LIN {X 0,Y 200.13,Z 356.551,A -85,B 0,C 180,E1 -21501.925,E2 -21501.925} C_VEL
LIN {X 0,Y 200.321,Z 356.531,A -85,B 0,C 180,E1 -21507.99,E2 -21507.99} C_VEL
LIN {X 0,Y 200.478,Z 356.509,A -85,B 0,C 180,E1 -21510,E2 -21510} C_VEL
LIN {X 0,Y 200.031,Z 356.568,A -85,B 0,C 180,E1 -21514.03,E2 -21514.03} C_VEL
LIN {X 0,Y 200.13,Z 356.553,A -85,B 0,C 180,E1 -21518.075,E2 -21518.075} C_VEL
LIN {X 0,Y 199.913,Z 356.584,A -85,B 0,C 180,E1 -21522.177,E2 -21522.177} C_VEL
LIN {X 0,Y 199.803,Z 356.594,A -85,B 0,C 180,E1 -21526.344,E2 -21526.344} C_VEL
LIN {X 0,Y 199.698,Z 356.609,A -85,B 0,C 180,E1 -21530.606,E2 -21530.606} C_VEL
LIN {X 0,Y 199.671,Z 356.608,A -85,B 0,C 180,E1 -21534.985,E2 -21534.985} C_VEL
LIN {X 0,Y 199.663,Z 356.613,A -85,B 0,C 180,E1 -21539.525,E2 -21539.525} C_VEL
LIN {X 0,Y 199.657,Z 356.613,A -85,B 0,C 180,E1 -21542.35,E2 -21542.35} C_VEL
LIN {X 0,Y 199.639,Z 356.615,A -85,B 0,C 180,E1 -21546.76,E2 -21546.76} C_VEL
LIN {X 0,Y 199.638,Z 356.616,A -85,B 0,C 180,E1 -21549.322,E2 -21549.322} C_VEL
LIN {X 0,Y 199.58,Z 356.622,A -85,B 0,C 180,E1 -21554.772,E2 -21554.772} C_VEL
LIN {X 0,Y 199.58,Z 356.626,A -85,B 0,C 180,E1 -21558.006,E2 -21558.006} C_VEL
LIN {X 0,Y 199.641,Z 356.611,A -85,B 0,C 180,E1 -21560.758,E2 -21560.758} C_VEL
LIN {X 0,Y 199.738,Z 356.771,A -85,B 0,C 180,E1 -21564.401,E2 -21564.401} C_VEL
LIN {X 0,Y 207.724,Z 383.973,A -85,B 0,C 180,E1 -21566.367,E2 -21566.367} C_VEL
LIN {X 0,Y 205.676,Z 433.557,A -85,B 0,C 180,E1 -21569.071,E2 -21569.071} C_VEL
LIN {X 0,Y 205.054,Z 449.624,A -85,B 0,C 180,E1 -21570.131,E2 -21570.131} C_VEL
LIN {X 0,Y 204.201,Z 463.538,A -85,B 0,C 180,E1 -21571.477,E2 -21571.477} C_VEL
LIN {X 0,Y 203.276,Z 475.696,A -85,B 0,C 180,E1 -21573.015,E2 -21573.015} C_VEL
LIN {X 0,Y 202.255,Z 488.035,A -85,B 0,C 180,E1 -21575.007,E2 -21575.007} C_VEL
LIN {X 0,Y 201.181,Z 499.934,A -85,B 0,C 180,E1 -21577.403,E2 -21577.403} C_VEL
LIN {X 0,Y 200.238,Z 510.281,A -85,B 0,C 180,E1 -21579.99,E2 -21579.99} C_VEL
LIN {X 0,Y 199.569,Z 519.169,A -85,B 0,C 180,E1 -21582.696,E2 -21582.696} C_VEL
LIN {X 0,Y 199.062,Z 527.201,A -85,B 0,C 180,E1 -21585.693,E2 -21585.693} C_VEL
LIN {X 0,Y 198.897,Z 534.007,A -85,B 0,C 180,E1 -21588.795,E2 -21588.795} C_VEL
LIN {X 0,Y 199.169,Z 539.493,A -85,B 0,C 180,E1 -21591.887,E2 -21591.887} C_VEL
LIN {X 0,Y 199.667,Z 543.756,A -85,B 0,C 180,E1 -21594.953,E2 -21594.953} C_VEL
LIN {X 0,Y 200.694,Z 546.982,A -85,B 0,C 180,E1 -21597.994,E2 -21597.994} C_VEL
LIN {X 0,Y 201.659,Z 548.585,A -85,B 0,C 180,E1 -21600.001,E2 -21600.001} C_VEL
LIN {X 0,Y 204.197,Z 550.567,A -85,B 0,C 180,E1 -21603.948,E2 -21603.948} C_VEL
LIN {X 0,Y 205.761,Z 550.967,A -85,B 0,C 180,E1 -21605.882,E2 -21605.882} C_VEL
LIN {X 0,Y 207.575,Z 550.921,A -85,B 0,C 180,E1 -21607.784,E2 -21607.784} C_VEL
LIN {X 0,Y 211.909,Z 549.645,A -85,B 0,C 180,E1 -21611.479,E2 -21611.479} C_VEL
LIN {X 0,Y 214.316,Z 548.421,A -85,B 0,C 180,E1 -21613.271,E2 -21613.271} C_VEL
LIN {X 0,Y 218.335,Z 545.769,A -85,B 0,C 180,E1 -21615.88,E2 -21615.88} C_VEL
LIN {X 0,Y 224.368,Z 540.635,A -85,B 0,C 180,E1 -21619.203,E2 -21619.203} C_VEL
LIN {X 0,Y 230.212,Z 534.494,A -85,B 0,C 180,E1 -21621.962,E2 -21621.962} C_VEL
LIN {X 0,Y 235.618,Z 527.868,A -85,B 0,C 180,E1 -21624.214,E2 -21624.214} C_VEL
LIN {X 0,Y 241.34,Z 519.724,A -85,B 0,C 180,E1 -21626.366,E2 -21626.366} C_VEL
LIN {X 0,Y 247.352,Z 509.665,A -85,B 0,C 180,E1 -21628.42,E2 -21628.42} C_VEL
LIN {X 0,Y 252.531,Z 499.378,A -85,B 0,C 180,E1 -21630.063,E2 -21630.063} C_VEL
LIN {X 0,Y 257.926,Z 486.52,A -85,B 0,C 180,E1 -21631.637,E2 -21631.637} C_VEL
LIN {X 0,Y 262.112,Z 473.808,A -85,B 0,C 180,E1 -21632.857,E2 -21632.857} C_VEL
LIN {X 0,Y 265.465,Z 460.103,A -85,B 0,C 180,E1 -21633.86,E2 -21633.86} C_VEL
LIN {X 0,Y 269.789,Z 438.336,A -85,B 0,C 180,E1 -21635.008,E2 -21635.008} C_VEL
LIN {X 0,Y 269.332,Z 436.976,A -85,B 0,C 180,E1 -21636.008,E2 -21636.008} C_VEL
LIN {X 0,Y 268.866,Z 435.366,A -85,B 0,C 180,E1 -21637.692,E2 -21637.692} C_VEL
LIN {X 0,Y 268.411,Z 435.595,A -85,B 0,C 180,E1 -21639.946,E2 -21639.946} C_VEL
LIN {X 0,Y 268.781,Z 437.514,A -85,B 0,C 180,E1 -21642.832,E2 -21642.832} C_VEL
LIN {X 0,Y 268.989,Z 439.1,A -85,B 0,C 180,E1 -21643.838,E2 -21643.838} C_VEL
LIN {X 0,Y 266.129,Z 456.669,A -85,B 0,C 180,E1 -21645.491,E2 -21645.491} C_VEL
LIN {X 0,Y 265.42,Z 460.479,A -85,B 0,C 180,E1 -21645.712,E2 -21645.712} C_VEL
LIN {X 0,Y 264.093,Z 466.352,A -85,B 0,C 180,E1 -21645.82,E2 -21645.82} C_VEL
LIN {X 0,Y 259.559,Z 481.708,A -85,B 0,C 180,E1 -21645.699,E2 -21645.699} C_VEL
LIN {X 0,Y 257.716,Z 487.218,A -85,B 0,C 180,E1 -21645.861,E2 -21645.861} C_VEL
LIN {X 0,Y 252.173,Z 502.361,A -85,B 0,C 180,E1 -21646.81,E2 -21646.81} C_VEL
LIN {X 0,Y 246.736,Z 514.517,A -85,B 0,C 180,E1 -21647.816,E2 -21647.816} C_VEL
LIN {X 0,Y 240.342,Z 526.637,A -85,B 0,C 180,E1 -21649.134,E2 -21649.134} C_VEL
LIN {X 0,Y 233.392,Z 538.193,A -85,B 0,C 180,E1 -21650.775,E2 -21650.775} C_VEL
LIN {X 0,Y 226.298,Z 548.528,A -85,B 0,C 180,E1 -21652.727,E2 -21652.727} C_VEL
LIN {X 0,Y 219.772,Z 557.196,A -85,B 0,C 180,E1 -21654.857,E2 -21654.857} C_VEL
LIN {X 0,Y 212.934,Z 565.506,A -85,B 0,C 180,E1 -21657.565,E2 -21657.565} C_VEL
LIN {X 0,Y 207.028,Z 572.262,A -85,B 0,C 180,E1 -21660.512,E2 -21660.512} C_VEL
LIN {X 0,Y 201.244,Z 578.3,A -85,B 0,C 180,E1 -21664.116,E2 -21664.116} C_VEL
LIN {X 0,Y 197.743,Z 581.793,A -85,B 0,C 180,E1 -21666.986,E2 -21666.986} C_VEL
LIN {X 0,Y 194.328,Z 585.191,A -85,B 0,C 180,E1 -21671.004,E2 -21671.004} C_VEL
LIN {X 0,Y 192.114,Z 587.173,A -85,B 0,C 180,E1 -21675.162,E2 -21675.162} C_VEL
LIN {X 0,Y 191.331,Z 587.716,A -85,B 0,C 180,E1 -21679.417,E2 -21679.417} C_VEL
LIN {X 0,Y 191.839,Z 586.864,A -85,B 0,C 180,E1 -21683.69,E2 -21683.69} C_VEL
LIN {X 0,Y 192.41,Z 585.854,A -85,B 0,C 180,E1 -21685.81,E2 -21685.81} C_VEL
LIN {X 0,Y 193.156,Z 584.419,A -85,B 0,C 180,E1 -21687.914,E2 -21687.914} C_VEL
LIN {X 0,Y 194.107,Z 581.798,A -85,B 0,C 180,E1 -21690.778,E2 -21690.778} C_VEL
LIN {X 0,Y 192.821,Z 584.818,A -85,B 0,C 180,E1 -21694.18,E2 -21694.18} C_VEL
LIN {X 0,Y 191.765,Z 586.935,A -85,B 0,C 180,E1 -21698.429,E2 -21698.429} C_VEL
LIN {X 0,Y 191.724,Z 587.605,A -85,B 0,C 180,E1 -21702.705,E2 -21702.705} C_VEL
LIN {X 0,Y 193.151,Z 586.968,A -85,B 0,C 180,E1 -21706.923,E2 -21706.923} C_VEL
LIN {X 0,Y 196.036,Z 584.878,A -85,B 0,C 180,E1 -21711.231,E2 -21711.231} C_VEL
LIN {X 0,Y 200.066,Z 581.723,A -85,B 0,C 180,E1 -21714.932,E2 -21714.932} C_VEL
LIN {X 0,Y 205.555,Z 577.043,A -85,B 0,C 180,E1 -21718.598,E2 -21718.598} C_VEL
LIN {X 0,Y 212.272,Z 570.882,A -85,B 0,C 180,E1 -21721.987,E2 -21721.987} C_VEL
LIN {X 0,Y 219.024,Z 564.138,A -85,B 0,C 180,E1 -21724.719,E2 -21724.719} C_VEL
LIN {X 0,Y 226.551,Z 555.909,A -85,B 0,C 180,E1 -21727.223,E2 -21727.223} C_VEL
LIN {X 0,Y 233.695,Z 547.449,A -85,B 0,C 180,E1 -21729.164,E2 -21729.164} C_VEL
LIN {X 0,Y 241.357,Z 537.432,A -85,B 0,C 180,E1 -21730.934,E2 -21730.934} C_VEL
LIN {X 0,Y 249.417,Z 525.489,A -85,B 0,C 180,E1 -21732.552,E2 -21732.552} C_VEL
LIN {X 0,Y 256.63,Z 513.371,A -85,B 0,C 180,E1 -21733.748,E2 -21733.748} C_VEL
LIN {X 0,Y 263.345,Z 500.187,A -85,B 0,C 180,E1 -21734.739,E2 -21734.739} C_VEL
LIN {X 0,Y 269.568,Z 485.453,A -85,B 0,C 180,E1 -21735.585,E2 -21735.585} C_VEL
LIN {X 0,Y 274.038,Z 472.123,A -85,B 0,C 180,E1 -21736.246,E2 -21736.246} C_VEL
LIN {X 0,Y 276.158,Z 464.301,A -85,B 0,C 180,E1 -21736.993,E2 -21736.993} C_VEL
LIN {X 0,Y 276.362,Z 463.489,A -85,B 0,C 180,E1 -21737.517,E2 -21737.517} C_VEL
LIN {X 0,Y 276.331,Z 463.603,A -85,B 0,C 180,E1 -21737.696,E2 -21737.696} C_VEL
LIN {X 0,Y 272.737,Z 475.349,A -85,B 0,C 180,E1 -21738.477,E2 -21738.477} C_VEL
LIN {X 0,Y 268.039,Z 487.452,A -85,B 0,C 180,E1 -21739.498,E2 -21739.498} C_VEL
LIN {X 0,Y 262.451,Z 499.125,A -85,B 0,C 180,E1 -21740.754,E2 -21740.754} C_VEL
LIN {X 0,Y 257,Z 508.731,A -85,B 0,C 180,E1 -21742.026,E2 -21742.026} C_VEL
LIN {X 0,Y 249.982,Z 519.179,A -85,B 0,C 180,E1 -21743.814,E2 -21743.814} C_VEL
LIN {X 0,Y 243.171,Z 527.827,A -85,B 0,C 180,E1 -21745.695,E2 -21745.695} C_VEL
LIN {X 0,Y 235.644,Z 535.955,A -85,B 0,C 180,E1 -21748.035,E2 -21748.035} C_VEL
LIN {X 0,Y 228.609,Z 542.34,A -85,B 0,C 180,E1 -21750.535,E2 -21750.535} C_VEL
LIN {X 0,Y 222.953,Z 546.638,A -85,B 0,C 180,E1 -21752.801,E2 -21752.801} C_VEL
LIN {X 0,Y 217.696,Z 549.945,A -85,B 0,C 180,E1 -21755.184,E2 -21755.184} C_VEL
LIN {X 0,Y 211.361,Z 552.899,A -85,B 0,C 180,E1 -21758.545,E2 -21758.545} C_VEL
LIN {X 0,Y 208.492,Z 553.807,A -85,B 0,C 180,E1 -21760.3,E2 -21760.3} C_VEL
LIN {X 0,Y 203.337,Z 554.428,A -85,B 0,C 180,E1 -21763.947,E2 -21763.947} C_VEL
LIN {X 0,Y 199.159,Z 553.524,A -85,B 0,C 180,E1 -21767.775,E2 -21767.775} C_VEL
LIN {X 0,Y 197.465,Z 552.5,A -85,B 0,C 180,E1 -21769.748,E2 -21769.748} C_VEL
LIN {X 0,Y 194.698,Z 549.233,A -85,B 0,C 180,E1 -21773.782,E2 -21773.782} C_VEL
LIN {X 0,Y 192.883,Z 544.368,A -85,B 0,C 180,E1 -21777.911,E2 -21777.911} C_VEL
LIN {X 0,Y 192.027,Z 539.501,A -85,B 0,C 180,E1 -21781.048,E2 -21781.048} C_VEL
LIN {X 0,Y 191.753,Z 532.354,A -85,B 0,C 180,E1 -21784.729,E2 -21784.729} C_VEL
LIN {X 0,Y 191.932,Z 526.232,A -85,B 0,C 180,E1 -21787.335,E2 -21787.335} C_VEL
LIN {X 0,Y 192.376,Z 517.232,A -85,B 0,C 180,E1 -21790.524,E2 -21790.524} C_VEL
LIN {X 0,Y 193.015,Z 507.213,A -85,B 0,C 180,E1 -21793.421,E2 -21793.421} C_VEL
LIN {X 0,Y 193.977,Z 494.938,A -85,B 0,C 180,E1 -21796.306,E2 -21796.306} C_VEL
LIN {X 0,Y 194.877,Z 482.252,A -85,B 0,C 180,E1 -21798.666,E2 -21798.666} C_VEL
LIN {X 0,Y 195.949,Z 469.152,A -85,B 0,C 180,E1 -21800.605,E2 -21800.605} C_VEL
LIN {X 0,Y 196.739,Z 454.506,A -85,B 0,C 180,E1 -21802.263,E2 -21802.263} C_VEL
LIN {X 0,Y 197.458,Z 440.483,A -85,B 0,C 180,E1 -21803.395,E2 -21803.395} C_VEL
LIN {X 0,Y 199.499,Z 382.365,A -85,B 0,C 180,E1 -21806.992,E2 -21806.992} C_VEL
LIN {X 0,Y 192.727,Z 357.475,A -85,B 0,C 180,E1 -21808.874,E2 -21808.874} C_VEL
LIN {X 0,Y 192.598,Z 357.494,A -85,B 0,C 180,E1 -21813.185,E2 -21813.185} C_VEL
LIN {X 0,Y 192.55,Z 357.496,A -85,B 0,C 180,E1 -21818.351,E2 -21818.351} C_VEL
LIN {X 0,Y 192.49,Z 357.507,A -85,B 0,C 180,E1 -21823.095,E2 -21823.095} C_VEL
LIN {X 0,Y 192.513,Z 357.501,A -85,B 0,C 180,E1 -21826.896,E2 -21826.896} C_VEL
LIN {X 0,Y 192.572,Z 357.496,A -85,B 0,C 180,E1 -21831.653,E2 -21831.653} C_VEL
LIN {X 0,Y 192.596,Z 357.493,A -85,B 0,C 180,E1 -21834.278,E2 -21834.278} C_VEL
LIN {X 0,Y 192.597,Z 357.493,A -85,B 0,C 180,E1 -21839.278,E2 -21839.278} C_VEL
LIN {X 0,Y 192.658,Z 357.484,A -85,B 0,C 180,E1 -21841.691,E2 -21841.691} C_VEL
LIN {X 0,Y 192.703,Z 357.479,A -85,B 0,C 180,E1 -21846.349,E2 -21846.349} C_VEL
LIN {X 0,Y 192.729,Z 357.474,A -85,B 0,C 180,E1 -21851.457,E2 -21851.457} C_VEL
LIN {X 0,Y 192.77,Z 357.471,A -85,B 0,C 180,E1 -21855.214,E2 -21855.214} C_VEL
LIN {X 0,Y 193.018,Z 357.439,A -85,B 0,C 180,E1 -21859.511,E2 -21859.511} C_VEL
LIN {X 0,Y 193.003,Z 357.441,A -85,B 0,C 180,E1 -21863.729,E2 -21863.729} C_VEL
LIN {X 0,Y 193.263,Z 357.41,A -85,B 0,C 180,E1 -21867.916,E2 -21867.916} C_VEL
LIN {X 0,Y 193.442,Z 357.385,A -85,B 0,C 180,E1 -21870,E2 -21870} C_VEL
LIN {X 0,Y 192.978,Z 357.447,A -85,B 0,C 180,E1 -21874.177,E2 -21874.177} C_VEL
LIN {X 0,Y 193.077,Z 357.431,A -85,B 0,C 180,E1 -21878.372,E2 -21878.372} C_VEL
LIN {X 0,Y 192.852,Z 357.462,A -85,B 0,C 180,E1 -21882.63,E2 -21882.63} C_VEL
LIN {X 0,Y 192.756,Z 357.469,A -85,B 0,C 180,E1 -21886.959,E2 -21886.959} C_VEL
LIN {X 0,Y 192.635,Z 357.488,A -85,B 0,C 180,E1 -21891.398,E2 -21891.398} C_VEL
LIN {X 0,Y 192.663,Z 357.484,A -85,B 0,C 180,E1 -21894.225,E2 -21894.225} C_VEL
LIN {X 0,Y 192.643,Z 357.487,A -85,B 0,C 180,E1 -21898.89,E2 -21898.89} C_VEL
LIN {X 0,Y 192.597,Z 357.49,A -85,B 0,C 180,E1 -21903.187,E2 -21903.187} C_VEL
LIN {X 0,Y 192.609,Z 357.492,A -85,B 0,C 180,E1 -21906.609,E2 -21906.609} C_VEL
LIN {X 0,Y 192.523,Z 357.5,A -85,B 0,C 180,E1 -21911.079,E2 -21911.079} C_VEL
LIN {X 0,Y 192.512,Z 357.506,A -85,B 0,C 180,E1 -21916.083,E2 -21916.083} C_VEL
LIN {X 0,Y 192.54,Z 357.499,A -85,B 0,C 180,E1 -21920.044,E2 -21920.044} C_VEL
LIN {X 0,Y 192.649,Z 357.488,A -85,B 0,C 180,E1 -21923.981,E2 -21923.981} C_VEL
LIN {X 0,Y 200.688,Z 384.623,A -85,B 0,C 180,E1 -21926.079,E2 -21926.079} C_VEL
LIN {X 0,Y 198.622,Z 434.427,A -85,B 0,C 180,E1 -21928.911,E2 -21928.911} C_VEL
LIN {X 0,Y 197.991,Z 450.137,A -85,B 0,C 180,E1 -21929.983,E2 -21929.983} C_VEL
LIN {X 0,Y 197.112,Z 464.132,A -85,B 0,C 180,E1 -21931.374,E2 -21931.374} C_VEL
LIN {X 0,Y 196.156,Z 476.48,A -85,B 0,C 180,E1 -21932.99,E2 -21932.99} C_VEL
LIN {X 0,Y 195.142,Z 488.274,A -85,B 0,C 180,E1 -21934.966,E2 -21934.966} C_VEL
LIN {X 0,Y 194.09,Z 499.915,A -85,B 0,C 180,E1 -21937.374,E2 -21937.374} C_VEL
LIN {X 0,Y 193.057,Z 511.324,A -85,B 0,C 180,E1 -21940.323,E2 -21940.323} C_VEL
LIN {X 0,Y 192.414,Z 519.875,A -85,B 0,C 180,E1 -21943.011,E2 -21943.011} C_VEL
LIN {X 0,Y 191.935,Z 528.245,A -85,B 0,C 180,E1 -21946.232,E2 -21946.232} C_VEL
LIN {X 0,Y 191.846,Z 535.03,A -85,B 0,C 180,E1 -21949.447,E2 -21949.447} C_VEL
LIN {X 0,Y 192.176,Z 540.475,A -85,B 0,C 180,E1 -21952.647,E2 -21952.647} C_VEL
LIN {X 0,Y 192.784,Z 544.764,A -85,B 0,C 180,E1 -21955.82,E2 -21955.82} C_VEL
LIN {X 0,Y 193.516,Z 547.04,A -85,B 0,C 180,E1 -21957.92,E2 -21957.92} C_VEL
LIN {X 0,Y 194.508,Z 548.879,A -85,B 0,C 180,E1 -21960.001,E2 -21960.001} C_VEL
LIN {X 0,Y 195.68,Z 550.312,A -85,B 0,C 180,E1 -21962.059,E2 -21962.059} C_VEL
LIN {X 0,Y 197.384,Z 551.462,A -85,B 0,C 180,E1 -21964.459,E2 -21964.459} C_VEL
LIN {X 0,Y 200.579,Z 552.142,A -85,B 0,C 180,E1 -21968.058,E2 -21968.058} C_VEL
LIN {X 0,Y 202.729,Z 551.962,A -85,B 0,C 180,E1 -21969.983,E2 -21969.983} C_VEL
LIN {X 0,Y 205.076,Z 551.368,A -85,B 0,C 180,E1 -21971.867,E2 -21971.867} C_VEL
LIN {X 0,Y 210.303,Z 548.958,A -85,B 0,C 180,E1 -21975.507,E2 -21975.507} C_VEL
LIN {X 0,Y 213.822,Z 546.747,A -85,B 0,C 180,E1 -21977.599,E2 -21977.599} C_VEL
LIN {X 0,Y 219.704,Z 542.124,A -85,B 0,C 180,E1 -21980.603,E2 -21980.603} C_VEL
LIN {X 0,Y 225.014,Z 537.117,A -85,B 0,C 180,E1 -21982.982,E2 -21982.982} C_VEL
LIN {X 0,Y 230.666,Z 530.851,A -85,B 0,C 180,E1 -21985.25,E2 -21985.25} C_VEL
LIN {X 0,Y 237.701,Z 521.712,A -85,B 0,C 180,E1 -21987.755,E2 -21987.755} C_VEL
LIN {X 0,Y 242.961,Z 513.651,A -85,B 0,C 180,E1 -21989.456,E2 -21989.456} C_VEL
LIN {X 0,Y 249.252,Z 502.412,A -85,B 0,C 180,E1 -21991.329,E2 -21991.329} C_VEL
LIN {X 0,Y 254.572,Z 490.786,A -85,B 0,C 180,E1 -21992.806,E2 -21992.806} C_VEL
LIN {X 0,Y 259.07,Z 478.805,A -85,B 0,C 180,E1 -21994.023,E2 -21994.023} C_VEL
LIN {X 0,Y 262.899,Z 465.581,A -85,B 0,C 180,E1 -21995.049,E2 -21995.049} C_VEL
LIN {X 0,Y 266.056,Z 450.737,A -85,B 0,C 180,E1 -21995.915,E2 -21995.915} C_VEL
LIN {X 0,Y 267.539,Z 443.724,A -85,B 0,C 180,E1 -21996.288,E2 -21996.288} C_VEL
LIN {X 0,Y 267.125,Z 442.24,A -85,B 0,C 180,E1 -21997.88,E2 -21997.88} C_VEL
LIN {X 0,Y 266.747,Z 442.503,A -85,B 0,C 180,E1 -21999.886,E2 -21999.886} C_VEL
LIN {X 0,Y 266.995,Z 444.365,A -85,B 0,C 180,E1 -22002.597,E2 -22002.597} C_VEL
LIN {X 0,Y 267.021,Z 444.576,A -85,B 0,C 180,E1 -22002.741,E2 -22002.741} C_VEL
LIN {X 0,Y 263.718,Z 462.474,A -85,B 0,C 180,E1 -22004.399,E2 -22004.399} C_VEL
LIN {X 0,Y 261.617,Z 473.4,A -85,B 0,C 180,E1 -22005.177,E2 -22005.177} C_VEL
LIN {X 0,Y 257.716,Z 487.218,A -85,B 0,C 180,E1 -22005.861,E2 -22005.861} C_VEL
LIN {X 0,Y 255.648,Z 492.809,A -85,B 0,C 180,E1 -22006.03,E2 -22006.03} C_VEL
LIN {X 0,Y 251.391,Z 501.746,A -85,B 0,C 180,E1 -22005.971,E2 -22005.971} C_VEL
LIN {X 0,Y 246.689,Z 510.398,A -85,B 0,C 180,E1 -22005.995,E2 -22005.995} C_VEL
LIN {X 0,Y 243.93,Z 515.393,A -85,B 0,C 180,E1 -22006.303,E2 -22006.303} C_VEL
LIN {X 0,Y 236.508,Z 528.466,A -85,B 0,C 180,E1 -22007.753,E2 -22007.753} C_VEL
LIN {X 0,Y 229.335,Z 539.311,A -85,B 0,C 180,E1 -22009.367,E2 -22009.367} C_VEL
LIN {X 0,Y 221.989,Z 549.224,A -85,B 0,C 180,E1 -22011.297,E2 -22011.297} C_VEL
LIN {X 0,Y 215.177,Z 557.482,A -85,B 0,C 180,E1 -22013.41,E2 -22013.41} C_VEL
LIN {X 0,Y 207.967,Z 565.461,A -85,B 0,C 180,E1 -22016.11,E2 -22016.11} C_VEL
LIN {X 0,Y 200.902,Z 572.726,A -85,B 0,C 180,E1 -22019.519,E2 -22019.519} C_VEL
LIN {X 0,Y 196.268,Z 577.061,A -85,B 0,C 180,E1 -22022.256,E2 -22022.256} C_VEL
LIN {X 0,Y 191.203,Z 581.517,A -85,B 0,C 180,E1 -22026.151,E2 -22026.151} C_VEL
LIN {X 0,Y 187.601,Z 584.519,A -85,B 0,C 180,E1 -22030.295,E2 -22030.295} C_VEL
LIN {X 0,Y 185.248,Z 586.153,A -85,B 0,C 180,E1 -22034.599,E2 -22034.599} C_VEL
LIN {X 0,Y 184.37,Z 586.445,A -85,B 0,C 180,E1 -22039.012,E2 -22039.012} C_VEL
LIN {X 0,Y 184.867,Z 585.307,A -85,B 0,C 180,E1 -22043.451,E2 -22043.451} C_VEL
LIN {X 0,Y 185.473,Z 584.166,A -85,B 0,C 180,E1 -22045.653,E2 -22045.653} C_VEL
LIN {X 0,Y 186.656,Z 581.612,A -85,B 0,C 180,E1 -22048.921,E2 -22048.921} C_VEL
LIN {X 0,Y 187.358,Z 579.59,A -85,B 0,C 180,E1 -22050.806,E2 -22050.806} C_VEL
LIN {X 0,Y 185.971,Z 582.827,A -85,B 0,C 180,E1 -22054.334,E2 -22054.334} C_VEL
LIN {X 0,Y 184.847,Z 585.245,A -85,B 0,C 180,E1 -22058.747,E2 -22058.747} C_VEL
LIN {X 0,Y 184.846,Z 586.225,A -85,B 0,C 180,E1 -22063.186,E2 -22063.186} C_VEL
LIN {X 0,Y 186.365,Z 585.91,A -85,B 0,C 180,E1 -22067.559,E2 -22067.559} C_VEL
LIN {X 0,Y 189.237,Z 584.289,A -85,B 0,C 180,E1 -22071.801,E2 -22071.801} C_VEL
LIN {X 0,Y 193.651,Z 581.401,A -85,B 0,C 180,E1 -22075.817,E2 -22075.817} C_VEL
LIN {X 0,Y 199.364,Z 577.196,A -85,B 0,C 180,E1 -22079.573,E2 -22079.573} C_VEL
LIN {X 0,Y 206.32,Z 571.582,A -85,B 0,C 180,E1 -22083.026,E2 -22083.026} C_VEL
LIN {X 0,Y 214.334,Z 564.352,A -85,B 0,C 180,E1 -22086.172,E2 -22086.172} C_VEL
LIN {X 0,Y 222.215,Z 556.563,A -85,B 0,C 180,E1 -22088.655,E2 -22088.655} C_VEL
LIN {X 0,Y 229.62,Z 548.574,A -85,B 0,C 180,E1 -22090.572,E2 -22090.572} C_VEL
LIN {X 0,Y 237.681,Z 538.972,A -85,B 0,C 180,E1 -22092.333,E2 -22092.333} C_VEL
LIN {X 0,Y 246.54,Z 526.919,A -85,B 0,C 180,E1 -22094.015,E2 -22094.015} C_VEL
LIN {X 0,Y 253.958,Z 515.491,A -85,B 0,C 180,E1 -22095.165,E2 -22095.165} C_VEL
LIN {X 0,Y 261.65,Z 501.585,A -85,B 0,C 180,E1 -22096.209,E2 -22096.209} C_VEL
LIN {X 0,Y 268.087,Z 487.622,A -85,B 0,C 180,E1 -22097.002,E2 -22097.002} C_VEL
LIN {X 0,Y 269.692,Z 483.656,A -85,B 0,C 180,E1 -22097.198,E2 -22097.198} C_VEL
LIN {X 0,Y 270.146,Z 482.401,A -85,B 0,C 180,E1 -22097.436,E2 -22097.436} C_VEL
LIN {X 0,Y 264.358,Z 495.071,A -85,B 0,C 180,E1 -22098.6,E2 -22098.6} C_VEL
LIN {X 0,Y 257.994,Z 506.481,A -85,B 0,C 180,E1 -22099.941,E2 -22099.941} C_VEL
LIN {X 0,Y 251.328,Z 516.468,A -85,B 0,C 180,E1 -22101.459,E2 -22101.459} C_VEL
LIN {X 0,Y 243.909,Z 525.948,A -85,B 0,C 180,E1 -22103.28,E2 -22103.28} C_VEL
LIN {X 0,Y 236.936,Z 533.527,A -85,B 0,C 180,E1 -22105.179,E2 -22105.179} C_VEL
LIN {X 0,Y 229.184,Z 540.728,A -85,B 0,C 180,E1 -22107.544,E2 -22107.544} C_VEL
LIN {X 0,Y 220.945,Z 546.965,A -85,B 0,C 180,E1 -22110.459,E2 -22110.459} C_VEL
LIN {X 0,Y 215.201,Z 550.488,A -85,B 0,C 180,E1 -22112.792,E2 -22112.792} C_VEL
LIN {X 0,Y 211.587,Z 552.337,A -85,B 0,C 180,E1 -22114.417,E2 -22114.417} C_VEL
LIN {X 0,Y 208.165,Z 553.761,A -85,B 0,C 180,E1 -22116.099,E2 -22116.099} C_VEL
LIN {X 0,Y 201.997,Z 555.423,A -85,B 0,C 180,E1 -22119.639,E2 -22119.639} C_VEL
LIN {X 0,Y 196.63,Z 555.631,A -85,B 0,C 180,E1 -22123.384,E2 -22123.384} C_VEL
LIN {X 0,Y 192.261,Z 554.259,A -85,B 0,C 180,E1 -22127.329,E2 -22127.329} C_VEL
LIN {X 0,Y 188.969,Z 551.386,A -85,B 0,C 180,E1 -22131.444,E2 -22131.444} C_VEL
LIN {X 0,Y 187.103,Z 548.173,A -85,B 0,C 180,E1 -22134.611,E2 -22134.611} C_VEL
LIN {X 0,Y 185.795,Z 544.013,A -85,B 0,C 180,E1 -22137.831,E2 -22137.831} C_VEL
LIN {X 0,Y 184.928,Z 538.801,A -85,B 0,C 180,E1 -22141.088,E2 -22141.088} C_VEL
LIN {X 0,Y 184.707,Z 531.242,A -85,B 0,C 180,E1 -22144.91,E2 -22144.91} C_VEL
LIN {X 0,Y 184.913,Z 523.993,A -85,B 0,C 180,E1 -22147.908,E2 -22147.908} C_VEL
LIN {X 0,Y 185.411,Z 515.207,A -85,B 0,C 180,E1 -22150.924,E2 -22150.924} C_VEL
LIN {X 0,Y 186.063,Z 504.602,A -85,B 0,C 180,E1 -22153.933,E2 -22153.933} C_VEL
LIN {X 0,Y 187.02,Z 492.722,A -85,B 0,C 180,E1 -22156.65,E2 -22156.65} C_VEL
LIN {X 0,Y 187.882,Z 481.063,A -85,B 0,C 180,E1 -22158.821,E2 -22158.821} C_VEL
LIN {X 0,Y 188.946,Z 467.407,A -85,B 0,C 180,E1 -22160.834,E2 -22160.834} C_VEL
LIN {X 0,Y 189.688,Z 453.534,A -85,B 0,C 180,E1 -22162.389,E2 -22162.389} C_VEL
LIN {X 0,Y 190.415,Z 439.593,A -85,B 0,C 180,E1 -22163.519,E2 -22163.519} C_VEL
LIN {X 0,Y 192.431,Z 383.401,A -85,B 0,C 180,E1 -22167.166,E2 -22167.166} C_VEL
LIN {X 0,Y 185.653,Z 358.355,A -85,B 0,C 180,E1 -22169.104,E2 -22169.104} C_VEL
LIN {X 0,Y 185.498,Z 358.379,A -85,B 0,C 180,E1 -22174.631,E2 -22174.631} C_VEL
LIN {X 0,Y 185.504,Z 358.374,A -85,B 0,C 180,E1 -22177.312,E2 -22177.312} C_VEL
LIN {X 0,Y 185.47,Z 358.381,A -85,B 0,C 180,E1 -22180.724,E2 -22180.724} C_VEL
LIN {X 0,Y 185.48,Z 358.377,A -85,B 0,C 180,E1 -22186.047,E2 -22186.047} C_VEL
LIN {X 0,Y 185.487,Z 358.378,A -85,B 0,C 180,E1 -22189.901,E2 -22189.901} C_VEL
LIN {X 0,Y 185.541,Z 358.373,A -85,B 0,C 180,E1 -22192.695,E2 -22192.695} C_VEL
LIN {X 0,Y 185.538,Z 358.371,A -85,B 0,C 180,E1 -22197.974,E2 -22197.974} C_VEL
LIN {X 0,Y 185.578,Z 358.37,A -85,B 0,C 180,E1 -22200.576,E2 -22200.576} C_VEL
LIN {X 0,Y 185.585,Z 358.364,A -85,B 0,C 180,E1 -22205.382,E2 -22205.382} C_VEL
LIN {X 0,Y 185.605,Z 358.364,A -85,B 0,C 180,E1 -22210.075,E2 -22210.075} C_VEL
LIN {X 0,Y 185.722,Z 358.35,A -85,B 0,C 180,E1 -22214.64,E2 -22214.64} C_VEL
LIN {X 0,Y 185.94,Z 358.32,A -85,B 0,C 180,E1 -22219.328,E2 -22219.328} C_VEL
LIN {X 0,Y 185.967,Z 358.317,A -85,B 0,C 180,E1 -22223.49,E2 -22223.49} C_VEL
LIN {X 0,Y 186.207,Z 358.288,A -85,B 0,C 180,E1 -22227.837,E2 -22227.837} C_VEL
LIN {X 0,Y 186.405,Z 358.261,A -85,B 0,C 180,E1 -22230,E2 -22230} C_VEL
LIN {X 0,Y 185.926,Z 358.327,A -85,B 0,C 180,E1 -22234.336,E2 -22234.336} C_VEL
LIN {X 0,Y 186.027,Z 358.309,A -85,B 0,C 180,E1 -22238.692,E2 -22238.692} C_VEL
LIN {X 0,Y 185.763,Z 358.344,A -85,B 0,C 180,E1 -22243.121,E2 -22243.121} C_VEL
LIN {X 0,Y 185.688,Z 358.349,A -85,B 0,C 180,E1 -22247.626,E2 -22247.626} C_VEL
LIN {X 0,Y 185.595,Z 358.367,A -85,B 0,C 180,E1 -22252.252,E2 -22252.252} C_VEL
LIN {X 0,Y 185.559,Z 358.368,A -85,B 0,C 180,E1 -22257.033,E2 -22257.033} C_VEL
LIN {X 0,Y 185.576,Z 358.368,A -85,B 0,C 180,E1 -22259.494,E2 -22259.494} C_VEL
LIN {X 0,Y 185.517,Z 358.373,A -85,B 0,C 180,E1 -22264.629,E2 -22264.629} C_VEL
LIN {X 0,Y 185.543,Z 358.371,A -85,B 0,C 180,E1 -22267.305,E2 -22267.305} C_VEL
LIN {X 0,Y 185.485,Z 358.377,A -85,B 0,C 180,E1 -22270.731,E2 -22270.731} C_VEL
LIN {X 0,Y 185.478,Z 358.382,A -85,B 0,C 180,E1 -22276.05,E2 -22276.05} C_VEL
LIN {X 0,Y 185.488,Z 358.378,A -85,B 0,C 180,E1 -22279.902,E2 -22279.902} C_VEL
LIN {X 0,Y 185.63,Z 358.433,A -85,B 0,C 180,E1 -22283.681,E2 -22283.681} C_VEL
LIN {X 0,Y 193.594,Z 386.068,A -85,B 0,C 180,E1 -22285.823,E2 -22285.823} C_VEL
LIN {X 0,Y 191.303,Z 441.155,A -85,B 0,C 180,E1 -22289.126,E2 -22289.126} C_VEL
LIN {X 0,Y 190.593,Z 455.398,A -85,B 0,C 180,E1 -22290.298,E2 -22290.298} C_VEL
LIN {X 0,Y 189.683,Z 469.139,A -85,B 0,C 180,E1 -22291.871,E2 -22291.871} C_VEL
LIN {X 0,Y 188.63,Z 481.707,A -85,B 0,C 180,E1 -22293.741,E2 -22293.741} C_VEL
LIN {X 0,Y 187.552,Z 493.474,A -85,B 0,C 180,E1 -22295.953,E2 -22295.953} C_VEL
LIN {X 0,Y 186.55,Z 504.298,A -85,B 0,C 180,E1 -22298.451,E2 -22298.451} C_VEL
LIN {X 0,Y 185.707,Z 514.647,A -85,B 0,C 180,E1 -22301.38,E2 -22301.38} C_VEL
LIN {X 0,Y 185.082,Z 523.842,A -85,B 0,C 180,E1 -22304.586,E2 -22304.586} C_VEL
LIN {X 0,Y 184.749,Z 531.604,A -85,B 0,C 180,E1 -22307.924,E2 -22307.924} C_VEL
LIN {X 0,Y 184.919,Z 537.913,A -85,B 0,C 180,E1 -22311.257,E2 -22311.257} C_VEL
LIN {X 0,Y 185.368,Z 542.985,A -85,B 0,C 180,E1 -22314.562,E2 -22314.562} C_VEL
LIN {X 0,Y 186.341,Z 546.938,A -85,B 0,C 180,E1 -22317.84,E2 -22317.84} C_VEL
LIN {X 0,Y 187.348,Z 549.033,A -85,B 0,C 180,E1 -22320.001,E2 -22320.001} C_VEL
LIN {X 0,Y 188.546,Z 550.705,A -85,B 0,C 180,E1 -22322.137,E2 -22322.137} C_VEL
LIN {X 0,Y 191.679,Z 552.789,A -85,B 0,C 180,E1 -22326.316,E2 -22326.316} C_VEL
LIN {X 0,Y 193.578,Z 553.264,A -85,B 0,C 180,E1 -22328.351,E2 -22328.351} C_VEL
LIN {X 0,Y 195.799,Z 553.306,A -85,B 0,C 180,E1 -22330.34,E2 -22330.34} C_VEL
LIN {X 0,Y 200.853,Z 552.197,A -85,B 0,C 180,E1 -22334.179,E2 -22334.179} C_VEL
LIN {X 0,Y 203.676,Z 551.088,A -85,B 0,C 180,E1 -22336.025,E2 -22336.025} C_VEL
LIN {X 0,Y 206.703,Z 549.524,A -85,B 0,C 180,E1 -22337.82,E2 -22337.82} C_VEL
LIN {X 0,Y 213.406,Z 545.132,A -85,B 0,C 180,E1 -22341.24,E2 -22341.24} C_VEL
LIN {X 0,Y 218.914,Z 540.596,A -85,B 0,C 180,E1 -22343.66,E2 -22343.66} C_VEL
LIN {X 0,Y 225.783,Z 533.837,A -85,B 0,C 180,E1 -22346.332,E2 -22346.332} C_VEL
LIN {X 0,Y 232.005,Z 526.651,A -85,B 0,C 180,E1 -22348.449,E2 -22348.449} C_VEL
LIN {X 0,Y 237.551,Z 519.283,A -85,B 0,C 180,E1 -22350.196,E2 -22350.196} C_VEL
LIN {X 0,Y 243.225,Z 510.52,A -85,B 0,C 180,E1 -22351.826,E2 -22351.826} C_VEL
LIN {X 0,Y 248.402,Z 501.222,A -85,B 0,C 180,E1 -22353.243,E2 -22353.243} C_VEL
LIN {X 0,Y 253.771,Z 489.827,A -85,B 0,C 180,E1 -22354.593,E2 -22354.593} C_VEL
LIN {X 0,Y 258.464,Z 477.26,A -85,B 0,C 180,E1 -22355.777,E2 -22355.777} C_VEL
LIN {X 0,Y 262.157,Z 464.532,A -85,B 0,C 180,E1 -22356.714,E2 -22356.714} C_VEL
LIN {X 0,Y 265.481,Z 449.693,A -85,B 0,C 180,E1 -22357.509,E2 -22357.509} C_VEL
LIN {X 0,Y 265.442,Z 449.187,A -85,B 0,C 180,E1 -22357.887,E2 -22357.887} C_VEL
LIN {X 0,Y 265.06,Z 449.569,A -85,B 0,C 180,E1 -22360.192,E2 -22360.192} C_VEL
LIN {X 0,Y 265.129,Z 450.526,A -85,B 0,C 180,E1 -22361.679,E2 -22361.679} C_VEL
LIN {X 0,Y 261.775,Z 467.097,A -85,B 0,C 180,E1 -22363.158,E2 -22363.158} C_VEL
LIN {X 0,Y 259.754,Z 475.532,A -85,B 0,C 180,E1 -22363.725,E2 -22363.725} C_VEL
LIN {X 0,Y 254.895,Z 490.692,A -85,B 0,C 180,E1 -22364.485,E2 -22364.485} C_VEL
LIN {X 0,Y 249.116,Z 504.885,A -85,B 0,C 180,E1 -22365.415,E2 -22365.415} C_VEL
LIN {X 0,Y 243.93,Z 515.393,A -85,B 0,C 180,E1 -22366.303,E2 -22366.303} C_VEL
LIN {X 0,Y 240.956,Z 520.437,A -85,B 0,C 180,E1 -22366.663,E2 -22366.663} C_VEL
LIN {X 0,Y 235.111,Z 528.541,A -85,B 0,C 180,E1 -22366.926,E2 -22366.926} C_VEL
LIN {X 0,Y 229.039,Z 535.975,A -85,B 0,C 180,E1 -22367.303,E2 -22367.303} C_VEL
LIN {X 0,Y 225.709,Z 540.172,A -85,B 0,C 180,E1 -22367.842,E2 -22367.842} C_VEL
LIN {X 0,Y 217.812,Z 549.934,A -85,B 0,C 180,E1 -22369.809,E2 -22369.809} C_VEL
LIN {X 0,Y 209.6,Z 559.015,A -85,B 0,C 180,E1 -22372.27,E2 -22372.27} C_VEL
LIN {X 0,Y 202.176,Z 566.394,A -85,B 0,C 180,E1 -22375,E2 -22375} C_VEL
LIN {X 0,Y 194.845,Z 573.116,A -85,B 0,C 180,E1 -22378.465,E2 -22378.465} C_VEL
LIN {X 0,Y 188.559,Z 578.26,A -85,B 0,C 180,E1 -22382.231,E2 -22382.231} C_VEL
LIN {X 0,Y 184.729,Z 581.125,A -85,B 0,C 180,E1 -22385.26,E2 -22385.26} C_VEL
LIN {X 0,Y 180.907,Z 583.802,A -85,B 0,C 180,E1 -22389.534,E2 -22389.534} C_VEL
LIN {X 0,Y 178.408,Z 585.093,A -85,B 0,C 180,E1 -22393.993,E2 -22393.993} C_VEL
LIN {X 0,Y 177.458,Z 585.048,A -85,B 0,C 180,E1 -22398.578,E2 -22398.578} C_VEL
LIN {X 0,Y 177.951,Z 583.656,A -85,B 0,C 180,E1 -22403.195,E2 -22403.195} C_VEL
LIN {X 0,Y 178.569,Z 582.391,A -85,B 0,C 180,E1 -22405.485,E2 -22405.485} C_VEL
LIN {X 0,Y 179.823,Z 579.659,A -85,B 0,C 180,E1 -22408.88,E2 -22408.88} C_VEL
LIN {X 0,Y 180.58,Z 577.465,A -85,B 0,C 180,E1 -22410.975,E2 -22410.975} C_VEL
LIN {X 0,Y 179.154,Z 580.759,A -85,B 0,C 180,E1 -22414.5,E2 -22414.5} C_VEL
LIN {X 0,Y 177.963,Z 583.466,A -85,B 0,C 180,E1 -22419.141,E2 -22419.141} C_VEL
LIN {X 0,Y 178.024,Z 584.705,A -85,B 0,C 180,E1 -22423.701,E2 -22423.701} C_VEL
LIN {X 0,Y 179.616,Z 584.708,A -85,B 0,C 180,E1 -22428.241,E2 -22428.241} C_VEL
LIN {X 0,Y 182.67,Z 583.465,A -85,B 0,C 180,E1 -22432.627,E2 -22432.627} C_VEL
LIN {X 0,Y 187.273,Z 581,A -85,B 0,C 180,E1 -22436.765,E2 -22436.765} C_VEL
LIN {X 0,Y 193.239,Z 577.259,A -85,B 0,C 180,E1 -22440.608,E2 -22440.608} C_VEL
LIN {X 0,Y 198.489,Z 573.54,A -85,B 0,C 180,E1 -22443.286,E2 -22443.286} C_VEL
LIN {X 0,Y 206.544,Z 567.35,A -85,B 0,C 180,E1 -22446.546,E2 -22446.546} C_VEL
LIN {X 0,Y 214.413,Z 560.602,A -85,B 0,C 180,E1 -22449.122,E2 -22449.122} C_VEL
LIN {X 0,Y 223.069,Z 552.381,A -85,B 0,C 180,E1 -22451.424,E2 -22451.424} C_VEL
LIN {X 0,Y 232.17,Z 542.74,A -85,B 0,C 180,E1 -22453.405,E2 -22453.405} C_VEL
LIN {X 0,Y 240.981,Z 532.204,A -85,B 0,C 180,E1 -22455.01,E2 -22455.01} C_VEL
LIN {X 0,Y 248.355,Z 522.198,A -85,B 0,C 180,E1 -22456.187,E2 -22456.187} C_VEL
LIN {X 0,Y 256.993,Z 508.814,A -85,B 0,C 180,E1 -22457.303,E2 -22457.303} C_VEL
LIN {X 0,Y 258.683,Z 505.859,A -85,B 0,C 180,E1 -22457.508,E2 -22457.508} C_VEL
LIN {X 0,Y 259.569,Z 504.177,A -85,B 0,C 180,E1 -22457.911,E2 -22457.911} C_VEL
LIN {X 0,Y 252.93,Z 514.202,A -85,B 0,C 180,E1 -22459.233,E2 -22459.233} C_VEL
LIN {X 0,Y 245.249,Z 524.046,A -85,B 0,C 180,E1 -22460.916,E2 -22460.916} C_VEL
LIN {X 0,Y 236.553,Z 533.401,A -85,B 0,C 180,E1 -22463.012,E2 -22463.012} C_VEL
LIN {X 0,Y 228.273,Z 540.801,A -85,B 0,C 180,E1 -22465.279,E2 -22465.279} C_VEL
LIN {X 0,Y 221.571,Z 545.877,A -85,B 0,C 180,E1 -22467.368,E2 -22467.368} C_VEL
LIN {X 0,Y 215.21,Z 549.927,A -85,B 0,C 180,E1 -22469.59,E2 -22469.59} C_VEL
LIN {X 0,Y 209.244,Z 553.022,A -85,B 0,C 180,E1 -22471.95,E2 -22471.95} C_VEL
LIN {X 0,Y 201.936,Z 555.768,A -85,B 0,C 180,E1 -22475.314,E2 -22475.314} C_VEL
LIN {X 0,Y 195.493,Z 556.955,A -85,B 0,C 180,E1 -22478.929,E2 -22478.929} C_VEL
LIN {X 0,Y 189.904,Z 556.671,A -85,B 0,C 180,E1 -22482.778,E2 -22482.778} C_VEL
LIN {X 0,Y 185.377,Z 554.892,A -85,B 0,C 180,E1 -22486.851,E2 -22486.851} C_VEL
LIN {X 0,Y 181.954,Z 551.547,A -85,B 0,C 180,E1 -22491.111,E2 -22491.111} C_VEL
LIN {X 0,Y 179.51,Z 546.653,A -85,B 0,C 180,E1 -22495.508,E2 -22495.508} C_VEL
LIN {X 0,Y 178.395,Z 541.807,A -85,B 0,C 180,E1 -22498.87,E2 -22498.87} C_VEL
LIN {X 0,Y 177.625,Z 534.701,A -85,B 0,C 180,E1 -22502.834,E2 -22502.834} C_VEL
LIN {X 0,Y 177.799,Z 527.286,A -85,B 0,C 180,E1 -22506.239,E2 -22506.239} C_VEL
LIN {X 0,Y 178.132,Z 518.728,A -85,B 0,C 180,E1 -22509.478,E2 -22509.478} C_VEL
LIN {X 0,Y 178.72,Z 508.066,A -85,B 0,C 180,E1 -22512.778,E2 -22512.778} C_VEL
LIN {X 0,Y 179.576,Z 496.867,A -85,B 0,C 180,E1 -22515.608,E2 -22515.608} C_VEL
LIN {X 0,Y 180.521,Z 484.396,A -85,B 0,C 180,E1 -22518.146,E2 -22518.146} C_VEL
LIN {X 0,Y 181.447,Z 472.498,A -85,B 0,C 180,E1 -22520.105,E2 -22520.105} C_VEL
LIN {X 0,Y 182.308,Z 459.356,A -85,B 0,C 180,E1 -22521.787,E2 -22521.787} C_VEL
LIN {X 0,Y 183.126,Z 444.972,A -85,B 0,C 180,E1 -22523.163,E2 -22523.163} C_VEL
LIN {X 0,Y 185.318,Z 384.323,A -85,B 0,C 180,E1 -22527.329,E2 -22527.329} C_VEL
LIN {X 0,Y 178.63,Z 359.476,A -85,B 0,C 180,E1 -22529.295,E2 -22529.295} C_VEL
LIN {X 0,Y 178.586,Z 359.233,A -85,B 0,C 180,E1 -22529.53,E2 -22529.53} C_VEL
LIN {X 0,Y 178.484,Z 359.251,A -85,B 0,C 180,E1 -22534.219,E2 -22534.219} C_VEL
LIN {X 0,Y 178.394,Z 359.261,A -85,B 0,C 180,E1 -22539.073,E2 -22539.073} C_VEL
LIN {X 0,Y 178.397,Z 359.262,A -85,B 0,C 180,E1 -22542.044,E2 -22542.044} C_VEL
LIN {X 0,Y 178.401,Z 359.26,A -85,B 0,C 180,E1 -22545.16,E2 -22545.16} C_VEL
LIN {X 0,Y 178.413,Z 359.258,A -85,B 0,C 180,E1 -22548.454,E2 -22548.454} C_VEL
LIN {X 0,Y 178.462,Z 359.254,A -85,B 0,C 180,E1 -22551.962,E2 -22551.962} C_VEL
LIN {X 0,Y 178.487,Z 359.248,A -85,B 0,C 180,E1 -22556.547,E2 -22556.547} C_VEL
LIN {X 0,Y 178.519,Z 359.247,A -85,B 0,C 180,E1 -22560.007,E2 -22560.007} C_VEL
LIN {X 0,Y 178.532,Z 359.244,A -85,B 0,C 180,E1 -22564.875,E2 -22564.875} C_VEL
LIN {X 0,Y 178.621,Z 359.233,A -85,B 0,C 180,E1 -22570.784,E2 -22570.784} C_VEL
LIN {X 0,Y 178.663,Z 359.226,A -85,B 0,C 180,E1 -22574.017,E2 -22574.017} C_VEL
LIN {X 0,Y 178.892,Z 359.199,A -85,B 0,C 180,E1 -22579.153,E2 -22579.153} C_VEL
LIN {X 0,Y 178.932,Z 359.194,A -85,B 0,C 180,E1 -22583.233,E2 -22583.233} C_VEL
LIN {X 0,Y 179.153,Z 359.167,A -85,B 0,C 180,E1 -22587.752,E2 -22587.752} C_VEL
LIN {X 0,Y 179.368,Z 359.137,A -85,B 0,C 180,E1 -22590,E2 -22590} C_VEL
LIN {X 0,Y 178.875,Z 359.204,A -85,B 0,C 180,E1 -22594.507,E2 -22594.507} C_VEL
LIN {X 0,Y 178.976,Z 359.186,A -85,B 0,C 180,E1 -22599.037,E2 -22599.037} C_VEL
LIN {X 0,Y 178.685,Z 359.226,A -85,B 0,C 180,E1 -22603.65,E2 -22603.65} C_VEL
LIN {X 0,Y 178.648,Z 359.23,A -85,B 0,C 180,E1 -22608.344,E2 -22608.344} C_VEL
LIN {X 0,Y 178.509,Z 359.247,A -85,B 0,C 180,E1 -22613.186,E2 -22613.186} C_VEL
LIN {X 0,Y 178.485,Z 359.252,A -85,B 0,C 180,E1 -22618.198,E2 -22618.198} C_VEL
LIN {X 0,Y 178.475,Z 359.252,A -85,B 0,C 180,E1 -22620.792,E2 -22620.792} C_VEL
LIN {X 0,Y 178.494,Z 359.247,A -85,B 0,C 180,E1 -22624.225,E2 -22624.225} C_VEL
LIN {X 0,Y 178.418,Z 359.259,A -85,B 0,C 180,E1 -22629.069,E2 -22629.069} C_VEL
LIN {X 0,Y 178.403,Z 359.259,A -85,B 0,C 180,E1 -22632.045,E2 -22632.045} C_VEL
LIN {X 0,Y 178.401,Z 359.26,A -85,B 0,C 180,E1 -22635.163,E2 -22635.163} C_VEL
LIN {X 0,Y 178.41,Z 359.26,A -85,B 0,C 180,E1 -22638.458,E2 -22638.458} C_VEL
LIN {X 0,Y 178.594,Z 359.429,A -85,B 0,C 180,E1 -22643.339,E2 -22643.339} C_VEL
LIN {X 0,Y 186.499,Z 386.513,A -85,B 0,C 180,E1 -22645.524,E2 -22645.524} C_VEL
LIN {X 0,Y 184.056,Z 445.577,A -85,B 0,C 180,E1 -22649.29,E2 -22649.29} C_VEL
LIN {X 0,Y 183.293,Z 459.427,A -85,B 0,C 180,E1 -22650.577,E2 -22650.577} C_VEL
LIN {X 0,Y 182.178,Z 473.903,A -85,B 0,C 180,E1 -22652.425,E2 -22652.425} C_VEL
LIN {X 0,Y 181.014,Z 487.517,A -85,B 0,C 180,E1 -22654.719,E2 -22654.719} C_VEL
LIN {X 0,Y 179.902,Z 499.575,A -85,B 0,C 180,E1 -22657.309,E2 -22657.309} C_VEL
LIN {X 0,Y 178.896,Z 510.494,A -85,B 0,C 180,E1 -22660.223,E2 -22660.223} C_VEL
LIN {X 0,Y 178.209,Z 520.123,A -85,B 0,C 180,E1 -22663.387,E2 -22663.387} C_VEL
LIN {X 0,Y 177.718,Z 528.805,A -85,B 0,C 180,E1 -22666.858,E2 -22666.858} C_VEL
LIN {X 0,Y 177.784,Z 536.882,A -85,B 0,C 180,E1 -22670.903,E2 -22670.903} C_VEL
LIN {X 0,Y 178.217,Z 542.337,A -85,B 0,C 180,E1 -22674.343,E2 -22674.343} C_VEL
LIN {X 0,Y 179.163,Z 546.685,A -85,B 0,C 180,E1 -22677.753,E2 -22677.753} C_VEL
LIN {X 0,Y 180.162,Z 549.037,A -85,B 0,C 180,E1 -22680.001,E2 -22680.001} C_VEL
LIN {X 0,Y 182.896,Z 552.406,A -85,B 0,C 180,E1 -22684.409,E2 -22684.409} C_VEL
LIN {X 0,Y 184.597,Z 553.523,A -85,B 0,C 180,E1 -22686.559,E2 -22686.559} C_VEL
LIN {X 0,Y 186.571,Z 554.215,A -85,B 0,C 180,E1 -22688.667,E2 -22688.667} C_VEL
LIN {X 0,Y 191.354,Z 554.4,A -85,B 0,C 180,E1 -22692.732,E2 -22692.732} C_VEL
LIN {X 0,Y 194.105,Z 553.927,A -85,B 0,C 180,E1 -22694.683,E2 -22694.683} C_VEL
LIN {X 0,Y 200.168,Z 551.756,A -85,B 0,C 180,E1 -22698.422,E2 -22698.422} C_VEL
LIN {X 0,Y 205.282,Z 549.072,A -85,B 0,C 180,E1 -22701.069,E2 -22701.069} C_VEL
LIN {X 0,Y 212.821,Z 543.933,A -85,B 0,C 180,E1 -22704.381,E2 -22704.381} C_VEL
LIN {X 0,Y 218.91,Z 538.784,A -85,B 0,C 180,E1 -22706.71,E2 -22706.71} C_VEL
LIN {X 0,Y 226.654,Z 531.04,A -85,B 0,C 180,E1 -22709.298,E2 -22709.298} C_VEL
LIN {X 0,Y 233.285,Z 523.098,A -85,B 0,C 180,E1 -22711.311,E2 -22711.311} C_VEL
LIN {X 0,Y 240.418,Z 513.156,A -85,B 0,C 180,E1 -22713.238,E2 -22713.238} C_VEL
LIN {X 0,Y 246.461,Z 502.974,A -85,B 0,C 180,E1 -22714.773,E2 -22714.773} C_VEL
LIN {X 0,Y 252.135,Z 491.716,A -85,B 0,C 180,E1 -22716.097,E2 -22716.097} C_VEL
LIN {X 0,Y 256.932,Z 479.747,A -85,B 0,C 180,E1 -22717.219,E2 -22717.219} C_VEL
LIN {X 0,Y 261.229,Z 465.846,A -85,B 0,C 180,E1 -22718.228,E2 -22718.228} C_VEL
LIN {X 0,Y 263.598,Z 456.078,A -85,B 0,C 180,E1 -22718.774,E2 -22718.774} C_VEL
LIN {X 0,Y 263.377,Z 456.808,A -85,B 0,C 180,E1 -22720.603,E2 -22720.603} C_VEL
LIN {X 0,Y 260.013,Z 471.196,A -85,B 0,C 180,E1 -22721.852,E2 -22721.852} C_VEL
LIN {X 0,Y 258.327,Z 477.216,A -85,B 0,C 180,E1 -22722.236,E2 -22722.236} C_VEL
LIN {X 0,Y 253.241,Z 491.718,A -85,B 0,C 180,E1 -22722.948,E2 -22722.948} C_VEL
LIN {X 0,Y 247.213,Z 505.299,A -85,B 0,C 180,E1 -22723.83,E2 -22723.83} C_VEL
LIN {X 0,Y 240.586,Z 517.818,A -85,B 0,C 180,E1 -22724.895,E2 -22724.895} C_VEL
LIN {X 0,Y 232.815,Z 530.229,A -85,B 0,C 180,E1 -22726.327,E2 -22726.327} C_VEL
LIN {X 0,Y 225.709,Z 540.172,A -85,B 0,C 180,E1 -22727.842,E2 -22727.842} C_VEL
LIN {X 0,Y 222.244,Z 544.329,A -85,B 0,C 180,E1 -22728.455,E2 -22728.455} C_VEL
LIN {X 0,Y 212.443,Z 553.333,A -85,B 0,C 180,E1 -22729.502,E2 -22729.502} C_VEL
LIN {X 0,Y 206.875,Z 557.97,A -85,B 0,C 180,E1 -22730.34,E2 -22730.34} C_VEL
LIN {X 0,Y 204.442,Z 560.077,A -85,B 0,C 180,E1 -22730.949,E2 -22730.949} C_VEL
LIN {X 0,Y 196.466,Z 567.272,A -85,B 0,C 180,E1 -22733.825,E2 -22733.825} C_VEL
LIN {X 0,Y 188.842,Z 573.425,A -85,B 0,C 180,E1 -22737.34,E2 -22737.34} C_VEL
LIN {X 0,Y 183.82,Z 577.08,A -85,B 0,C 180,E1 -22740.196,E2 -22740.196} C_VEL
LIN {X 0,Y 178.284,Z 580.671,A -85,B 0,C 180,E1 -22744.302,E2 -22744.302} C_VEL
LIN {X 0,Y 174.25,Z 582.953,A -85,B 0,C 180,E1 -22748.715,E2 -22748.715} C_VEL
LIN {X 0,Y 171.606,Z 583.927,A -85,B 0,C 180,E1 -22753.34,E2 -22753.34} C_VEL
LIN {X 0,Y 170.555,Z 583.606,A -85,B 0,C 180,E1 -22758.11,E2 -22758.11} C_VEL
LIN {X 0,Y 171.035,Z 581.917,A -85,B 0,C 180,E1 -22762.919,E2 -22762.919} C_VEL
LIN {X 0,Y 171.7,Z 580.5,A -85,B 0,C 180,E1 -22765.304,E2 -22765.304} C_VEL
LIN {X 0,Y 173.041,Z 577.555,A -85,B 0,C 180,E1 -22768.836,E2 -22768.836} C_VEL
LIN {X 0,Y 173.905,Z 575.102,A -85,B 0,C 180,E1 -22771.085,E2 -22771.085} C_VEL
LIN {X 0,Y 172.399,Z 578.547,A -85,B 0,C 180,E1 -22774.676,E2 -22774.676} C_VEL
LIN {X 0,Y 171.134,Z 581.503,A -85,B 0,C 180,E1 -22779.454,E2 -22779.454} C_VEL
LIN {X 0,Y 171.229,Z 583.08,A -85,B 0,C 180,E1 -22784.256,E2 -22784.256} C_VEL
LIN {X 0,Y 172.913,Z 583.422,A -85,B 0,C 180,E1 -22788.975,E2 -22788.975} C_VEL
LIN {X 0,Y 176.146,Z 582.558,A -85,B 0,C 180,E1 -22793.515,E2 -22793.515} C_VEL
LIN {X 0,Y 180.962,Z 580.5,A -85,B 0,C 180,E1 -22797.777,E2 -22797.777} C_VEL
LIN {X 0,Y 187.171,Z 577.195,A -85,B 0,C 180,E1 -22801.714,E2 -22801.714} C_VEL
LIN {X 0,Y 194.605,Z 572.585,A -85,B 0,C 180,E1 -22805.298,E2 -22805.298} C_VEL
LIN {X 0,Y 203.155,Z 566.585,A -85,B 0,C 180,E1 -22808.513,E2 -22808.513} C_VEL
LIN {X 0,Y 211.473,Z 560.055,A -85,B 0,C 180,E1 -22811.023,E2 -22811.023} C_VEL
LIN {X 0,Y 220.542,Z 552.146,A -85,B 0,C 180,E1 -22813.246,E2 -22813.246} C_VEL
LIN {X 0,Y 230.005,Z 542.851,A -85,B 0,C 180,E1 -22815.131,E2 -22815.131} C_VEL
LIN {X 0,Y 239.113,Z 532.703,A -85,B 0,C 180,E1 -22816.673,E2 -22816.673} C_VEL
LIN {X 0,Y 246.744,Z 523.094,A -85,B 0,C 180,E1 -22817.779,E2 -22817.779} C_VEL
LIN {X 0,Y 247.973,Z 521.476,A -85,B 0,C 180,E1 -22817.925,E2 -22817.925} C_VEL
LIN {X 0,Y 248.824,Z 520.162,A -85,B 0,C 180,E1 -22818.297,E2 -22818.297} C_VEL
LIN {X 0,Y 240.567,Z 529.449,A -85,B 0,C 180,E1 -22820.004,E2 -22820.004} C_VEL
LIN {X 0,Y 232.849,Z 536.82,A -85,B 0,C 180,E1 -22821.776,E2 -22821.776} C_VEL
LIN {X 0,Y 225.446,Z 542.878,A -85,B 0,C 180,E1 -22823.679,E2 -22823.679} C_VEL
LIN {X 0,Y 218.38,Z 547.79,A -85,B 0,C 180,E1 -22825.722,E2 -22825.722} C_VEL
LIN {X 0,Y 211.664,Z 551.687,A -85,B 0,C 180,E1 -22827.909,E2 -22827.909} C_VEL
LIN {X 0,Y 207.393,Z 553.788,A -85,B 0,C 180,E1 -22829.448,E2 -22829.448} C_VEL
LIN {X 0,Y 199.417,Z 556.729,A -85,B 0,C 180,E1 -22832.731,E2 -22832.731} C_VEL
LIN {X 0,Y 192.273,Z 558.183,A -85,B 0,C 180,E1 -22836.291,E2 -22836.291} C_VEL
LIN {X 0,Y 185.998,Z 558.164,A -85,B 0,C 180,E1 -22840.118,E2 -22840.118} C_VEL
LIN {X 0,Y 180.729,Z 556.649,A -85,B 0,C 180,E1 -22844.203,E2 -22844.203} C_VEL
LIN {X 0,Y 176.595,Z 553.669,A -85,B 0,C 180,E1 -22848.521,E2 -22848.521} C_VEL
LIN {X 0,Y 173.52,Z 549.089,A -85,B 0,C 180,E1 -22853.02,E2 -22853.02} C_VEL
LIN {X 0,Y 171.627,Z 542.865,A -85,B 0,C 180,E1 -22857.652,E2 -22857.652} C_VEL
LIN {X 0,Y 170.682,Z 535.769,A -85,B 0,C 180,E1 -22861.769,E2 -22861.769} C_VEL
LIN {X 0,Y 170.747,Z 527.027,A -85,B 0,C 180,E1 -22865.905,E2 -22865.905} C_VEL
LIN {X 0,Y 171.132,Z 516.9,A -85,B 0,C 180,E1 -22869.727,E2 -22869.727} C_VEL
LIN {X 0,Y 171.781,Z 506.25,A -85,B 0,C 180,E1 -22873.003,E2 -22873.003} C_VEL
LIN {X 0,Y 172.799,Z 493.174,A -85,B 0,C 180,E1 -22876.236,E2 -22876.236} C_VEL
LIN {X 0,Y 173.649,Z 481.253,A -85,B 0,C 180,E1 -22878.584,E2 -22878.584} C_VEL
LIN {X 0,Y 174.742,Z 467.339,A -85,B 0,C 180,E1 -22880.757,E2 -22880.757} C_VEL
LIN {X 0,Y 175.543,Z 452.64,A -85,B 0,C 180,E1 -22882.479,E2 -22882.479} C_VEL
LIN {X 0,Y 176.294,Z 437.622,A -85,B 0,C 180,E1 -22883.726,E2 -22883.726} C_VEL
LIN {X 0,Y 178.181,Z 385.01,A -85,B 0,C 180,E1 -22887.494,E2 -22887.494} C_VEL
LIN {X 0,Y 171.632,Z 360.57,A -85,B 0,C 180,E1 -22889.506,E2 -22889.506} C_VEL
LIN {X 0,Y 171.544,Z 360.11,A -85,B 0,C 180,E1 -22889.59,E2 -22889.59} C_VEL
LIN {X 0,Y 171.391,Z 360.136,A -85,B 0,C 180,E1 -22895.034,E2 -22895.034} C_VEL
LIN {X 0,Y 171.356,Z 360.136,A -85,B 0,C 180,E1 -22898.807,E2 -22898.807} C_VEL
LIN {X 0,Y 171.323,Z 360.143,A -85,B 0,C 180,E1 -22904.215,E2 -22904.215} C_VEL
LIN {X 0,Y 171.346,Z 360.141,A -85,B 0,C 180,E1 -22908.985,E2 -22908.985} C_VEL
LIN {X 0,Y 171.411,Z 360.132,A -85,B 0,C 180,E1 -22912.047,E2 -22912.047} C_VEL
LIN {X 0,Y 171.407,Z 360.128,A -85,B 0,C 180,E1 -22915.086,E2 -22915.086} C_VEL
LIN {X 0,Y 171.445,Z 360.13,A -85,B 0,C 180,E1 -22920.534,E2 -22920.534} C_VEL
LIN {X 0,Y 171.455,Z 360.124,A -85,B 0,C 180,E1 -22925.802,E2 -22925.802} C_VEL
LIN {X 0,Y 171.577,Z 360.11,A -85,B 0,C 180,E1 -22930.872,E2 -22930.872} C_VEL
LIN {X 0,Y 171.607,Z 360.107,A -85,B 0,C 180,E1 -22935.776,E2 -22935.776} C_VEL
LIN {X 0,Y 171.908,Z 360.067,A -85,B 0,C 180,E1 -22940.589,E2 -22940.589} C_VEL
LIN {X 0,Y 171.824,Z 360.081,A -85,B 0,C 180,E1 -22945.308,E2 -22945.308} C_VEL
LIN {X 0,Y 172.331,Z 360.014,A -85,B 0,C 180,E1 -22950,E2 -22950} C_VEL
LIN {X 0,Y 171.824,Z 360.081,A -85,B 0,C 180,E1 -22954.693,E2 -22954.693} C_VEL
LIN {X 0,Y 171.908,Z 360.067,A -85,B 0,C 180,E1 -22959.412,E2 -22959.412} C_VEL
LIN {X 0,Y 171.608,Z 360.109,A -85,B 0,C 180,E1 -22964.225,E2 -22964.225} C_VEL
LIN {X 0,Y 171.543,Z 360.115,A -85,B 0,C 180,E1 -22969.563,E2 -22969.563} C_VEL
LIN {X 0,Y 171.467,Z 360.121,A -85,B 0,C 180,E1 -22975.617,E2 -22975.617} C_VEL
LIN {X 0,Y 171.438,Z 360.129,A -85,B 0,C 180,E1 -22980.587,E2 -22980.587} C_VEL
LIN {X 0,Y 171.404,Z 360.13,A -85,B 0,C 180,E1 -22985.033,E2 -22985.033} C_VEL
LIN {X 0,Y 171.379,Z 360.136,A -85,B 0,C 180,E1 -22988.818,E2 -22988.818} C_VEL
LIN {X 0,Y 171.325,Z 360.142,A -85,B 0,C 180,E1 -22994.217,E2 -22994.217} C_VEL
LIN {X 0,Y 171.344,Z 360.139,A -85,B 0,C 180,E1 -22998.985,E2 -22998.985} C_VEL
LIN {X 0,Y 171.481,Z 360.121,A -85,B 0,C 180,E1 -23002.892,E2 -23002.892} C_VEL
LIN {X 0,Y 179.429,Z 387.654,A -85,B 0,C 180,E1 -23005.275,E2 -23005.275} C_VEL
LIN {X 0,Y 176.869,Z 447.983,A -85,B 0,C 180,E1 -23009.314,E2 -23009.314} C_VEL
LIN {X 0,Y 176.024,Z 461.881,A -85,B 0,C 180,E1 -23010.72,E2 -23010.72} C_VEL
LIN {X 0,Y 175.006,Z 474.613,A -85,B 0,C 180,E1 -23012.452,E2 -23012.452} C_VEL
LIN {X 0,Y 173.971,Z 486.803,A -85,B 0,C 180,E1 -23014.583,E2 -23014.583} C_VEL
LIN {X 0,Y 172.844,Z 499.141,A -85,B 0,C 180,E1 -23017.278,E2 -23017.278} C_VEL
LIN {X 0,Y 171.782,Z 510.946,A -85,B 0,C 180,E1 -23020.503,E2 -23020.503} C_VEL
LIN {X 0,Y 171.04,Z 520.951,A -85,B 0,C 180,E1 -23023.899,E2 -23023.899} C_VEL
LIN {X 0,Y 170.595,Z 529.634,A -85,B 0,C 180,E1 -23027.51,E2 -23027.51} C_VEL
LIN {X 0,Y 170.729,Z 536.624,A -85,B 0,C 180,E1 -23031.101,E2 -23031.101} C_VEL
LIN {X 0,Y 171.343,Z 543.203,A -85,B 0,C 180,E1 -23035.296,E2 -23035.296} C_VEL
LIN {X 0,Y 172.464,Z 547.596,A -85,B 0,C 180,E1 -23038.834,E2 -23038.834} C_VEL
LIN {X 0,Y 174.25,Z 550.977,A -85,B 0,C 180,E1 -23042.313,E2 -23042.313} C_VEL
LIN {X 0,Y 176.564,Z 553.411,A -85,B 0,C 180,E1 -23045.663,E2 -23045.663} C_VEL
LIN {X 0,Y 179.549,Z 555.005,A -85,B 0,C 180,E1 -23049.009,E2 -23049.009} C_VEL
LIN {X 0,Y 184.479,Z 555.73,A -85,B 0,C 180,E1 -23053.214,E2 -23053.214} C_VEL
LIN {X 0,Y 190.364,Z 554.867,A -85,B 0,C 180,E1 -23057.18,E2 -23057.18} C_VEL
LIN {X 0,Y 193.612,Z 553.869,A -85,B 0,C 180,E1 -23059.069,E2 -23059.069} C_VEL
LIN {X 0,Y 200.792,Z 550.656,A -85,B 0,C 180,E1 -23062.646,E2 -23062.646} C_VEL
LIN {X 0,Y 206.733,Z 547.095,A -85,B 0,C 180,E1 -23065.148,E2 -23065.148} C_VEL
LIN {X 0,Y 214.495,Z 541.315,A -85,B 0,C 180,E1 -23068.012,E2 -23068.012} C_VEL
LIN {X 0,Y 222.049,Z 534.489,A -85,B 0,C 180,E1 -23070.426,E2 -23070.426} C_VEL
LIN {X 0,Y 229.119,Z 526.948,A -85,B 0,C 180,E1 -23072.467,E2 -23072.467} C_VEL
LIN {X 0,Y 235.263,Z 519.294,A -85,B 0,C 180,E1 -23074.065,E2 -23074.065} C_VEL
LIN {X 0,Y 242.697,Z 508.453,A -85,B 0,C 180,E1 -23075.852,E2 -23075.852} C_VEL
LIN {X 0,Y 249.16,Z 496.951,A -85,B 0,C 180,E1 -23077.272,E2 -23077.272} C_VEL
LIN {X 0,Y 254.808,Z 484.637,A -85,B 0,C 180,E1 -23078.485,E2 -23078.485} C_VEL
LIN {X 0,Y 259.275,Z 472.073,A -85,B 0,C 180,E1 -23079.433,E2 -23079.433} C_VEL
LIN {X 0,Y 260.204,Z 468.993,A -85,B 0,C 180,E1 -23079.648,E2 -23079.648} C_VEL
LIN {X 0,Y 260.23,Z 468.884,A -85,B 0,C 180,E1 -23080.023,E2 -23080.023} C_VEL
LIN {X 0,Y 257.434,Z 478.214,A -85,B 0,C 180,E1 -23080.688,E2 -23080.688} C_VEL
LIN {X 0,Y 251.794,Z 492.938,A -85,B 0,C 180,E1 -23081.398,E2 -23081.398} C_VEL
LIN {X 0,Y 244.821,Z 507.439,A -85,B 0,C 180,E1 -23082.336,E2 -23082.336} C_VEL
LIN {X 0,Y 238.008,Z 519.215,A -85,B 0,C 180,E1 -23083.352,E2 -23083.352} C_VEL
LIN {X 0,Y 229.896,Z 531.218,A -85,B 0,C 180,E1 -23084.748,E2 -23084.748} C_VEL
LIN {X 0,Y 221.658,Z 541.792,A -85,B 0,C 180,E1 -23086.4,E2 -23086.4} C_VEL
LIN {X 0,Y 213.797,Z 550.712,A -85,B 0,C 180,E1 -23088.266,E2 -23088.266} C_VEL
LIN {X 0,Y 206.434,Z 558.222,A -85,B 0,C 180,E1 -23090.331,E2 -23090.331} C_VEL
LIN {X 0,Y 204.442,Z 560.077,A -85,B 0,C 180,E1 -23090.949,E2 -23090.949} C_VEL
LIN {X 0,Y 201.718,Z 562.215,A -85,B 0,C 180,E1 -23091.537,E2 -23091.537} C_VEL
LIN {X 0,Y 191.232,Z 568.123,A -85,B 0,C 180,E1 -23092.853,E2 -23092.853} C_VEL
LIN {X 0,Y 188.515,Z 569.752,A -85,B 0,C 180,E1 -23093.564,E2 -23093.564} C_VEL
LIN {X 0,Y 188.156,Z 570.006,A -85,B 0,C 180,E1 -23093.712,E2 -23093.712} C_VEL
LIN {X 0,Y 181.114,Z 574.823,A -85,B 0,C 180,E1 -23097.094,E2 -23097.094} C_VEL
LIN {X 0,Y 174.626,Z 578.713,A -85,B 0,C 180,E1 -23101.121,E2 -23101.121} C_VEL
LIN {X 0,Y 169.593,Z 581.255,A -85,B 0,C 180,E1 -23105.518,E2 -23105.518} C_VEL
LIN {X 0,Y 166.092,Z 582.52,A -85,B 0,C 180,E1 -23110.213,E2 -23110.213} C_VEL
LIN {X 0,Y 164.086,Z 582.496,A -85,B 0,C 180,E1 -23115.108,E2 -23115.108} C_VEL
LIN {X 0,Y 163.718,Z 581.217,A -85,B 0,C 180,E1 -23120.112,E2 -23120.112} C_VEL
LIN {X 0,Y 164.85,Z 578.538,A -85,B 0,C 180,E1 -23125.108,E2 -23125.108} C_VEL
LIN {X 0,Y 166.29,Z 575.393,A -85,B 0,C 180,E1 -23128.789,E2 -23128.789} C_VEL
LIN {X 0,Y 167.242,Z 572.657,A -85,B 0,C 180,E1 -23131.204,E2 -23131.204} C_VEL
LIN {X 0,Y 165.687,Z 576.222,A -85,B 0,C 180,E1 -23134.866,E2 -23134.866} C_VEL
LIN {X 0,Y 164.374,Z 579.481,A -85,B 0,C 180,E1 -23139.847,E2 -23139.847} C_VEL
LIN {X 0,Y 164.49,Z 581.357,A -85,B 0,C 180,E1 -23144.854,E2 -23144.854} C_VEL
LIN {X 0,Y 166.268,Z 582.017,A -85,B 0,C 180,E1 -23149.764,E2 -23149.764} C_VEL
LIN {X 0,Y 169.682,Z 581.509,A -85,B 0,C 180,E1 -23154.468,E2 -23154.468} C_VEL
LIN {X 0,Y 174.721,Z 579.844,A -85,B 0,C 180,E1 -23158.861,E2 -23158.861} C_VEL
LIN {X 0,Y 181.167,Z 576.989,A -85,B 0,C 180,E1 -23162.895,E2 -23162.895} C_VEL
LIN {X 0,Y 188.877,Z 572.891,A -85,B 0,C 180,E1 -23166.537,E2 -23166.537} C_VEL
LIN {X 0,Y 197.696,Z 567.484,A -85,B 0,C 180,E1 -23169.784,E2 -23169.784} C_VEL
LIN {X 0,Y 207.505,Z 560.616,A -85,B 0,C 180,E1 -23172.639,E2 -23172.639} C_VEL
LIN {X 0,Y 216.891,Z 553.168,A -85,B 0,C 180,E1 -23174.811,E2 -23174.811} C_VEL
LIN {X 0,Y 225.526,Z 545.503,A -85,B 0,C 180,E1 -23176.465,E2 -23176.465} C_VEL
LIN {X 0,Y 235.957,Z 535.011,A -85,B 0,C 180,E1 -23178.127,E2 -23178.127} C_VEL
LIN {X 0,Y 237.19,Z 533.693,A -85,B 0,C 180,E1 -23178.304,E2 -23178.304} C_VEL
LIN {X 0,Y 237.898,Z 532.777,A -85,B 0,C 180,E1 -23178.644,E2 -23178.644} C_VEL
LIN {X 0,Y 230.57,Z 539.218,A -85,B 0,C 180,E1 -23180.2,E2 -23180.2} C_VEL
LIN {X 0,Y 222.853,Z 545.043,A -85,B 0,C 180,E1 -23182.037,E2 -23182.037} C_VEL
LIN {X 0,Y 215.407,Z 549.788,A -85,B 0,C 180,E1 -23184.035,E2 -23184.035} C_VEL
LIN {X 0,Y 206.037,Z 554.541,A -85,B 0,C 180,E1 -23186.922,E2 -23186.922} C_VEL
LIN {X 0,Y 197.385,Z 557.745,A -85,B 0,C 180,E1 -23190.1,E2 -23190.1} C_VEL
LIN {X 0,Y 189.497,Z 559.398,A -85,B 0,C 180,E1 -23193.572,E2 -23193.572} C_VEL
LIN {X 0,Y 182.538,Z 559.609,A -85,B 0,C 180,E1 -23197.354,E2 -23197.354} C_VEL
LIN {X 0,Y 176.505,Z 558.385,A -85,B 0,C 180,E1 -23201.424,E2 -23201.424} C_VEL
LIN {X 0,Y 171.615,Z 555.649,A -85,B 0,C 180,E1 -23205.775,E2 -23205.775} C_VEL
LIN {X 0,Y 167.933,Z 551.442,A -85,B 0,C 180,E1 -23210.362,E2 -23210.362} C_VEL
LIN {X 0,Y 165.914,Z 547.207,A -85,B 0,C 180,E1 -23213.92,E2 -23213.92} C_VEL
LIN {X 0,Y 164.548,Z 541.988,A -85,B 0,C 180,E1 -23217.551,E2 -23217.551} C_VEL
LIN {X 0,Y 163.636,Z 534.45,A -85,B 0,C 180,E1 -23221.845,E2 -23221.845} C_VEL
LIN {X 0,Y 163.748,Z 525.137,A -85,B 0,C 180,E1 -23226.158,E2 -23226.158} C_VEL
LIN {X 0,Y 164.157,Z 515.262,A -85,B 0,C 180,E1 -23229.859,E2 -23229.859} C_VEL
LIN {X 0,Y 164.818,Z 504.148,A -85,B 0,C 180,E1 -23233.248,E2 -23233.248} C_VEL
LIN {X 0,Y 165.782,Z 491.749,A -85,B 0,C 180,E1 -23236.31,E2 -23236.31} C_VEL
LIN {X 0,Y 166.692,Z 479.423,A -85,B 0,C 180,E1 -23238.751,E2 -23238.751} C_VEL
LIN {X 0,Y 167.732,Z 465.84,A -85,B 0,C 180,E1 -23240.863,E2 -23240.863} C_VEL
LIN {X 0,Y 168.525,Z 451.577,A -85,B 0,C 180,E1 -23242.542,E2 -23242.542} C_VEL
LIN {X 0,Y 169.282,Z 434.836,A -85,B 0,C 180,E1 -23243.935,E2 -23243.935} C_VEL
LIN {X 0,Y 171.058,Z 386.058,A -85,B 0,C 180,E1 -23247.618,E2 -23247.618} C_VEL
LIN {X 0,Y 164.597,Z 361.619,A -85,B 0,C 180,E1 -23249.703,E2 -23249.703} C_VEL
LIN {X 0,Y 164.487,Z 360.989,A -85,B 0,C 180,E1 -23249.799,E2 -23249.799} C_VEL
LIN {X 0,Y 164.328,Z 361.014,A -85,B 0,C 180,E1 -23255.65,E2 -23255.65} C_VEL
LIN {X 0,Y 164.289,Z 361.016,A -85,B 0,C 180,E1 -23259.915,E2 -23259.915} C_VEL
LIN {X 0,Y 164.277,Z 361.021,A -85,B 0,C 180,E1 -23263.341,E2 -23263.341} C_VEL
LIN {X 0,Y 164.29,Z 361.016,A -85,B 0,C 180,E1 -23266.808,E2 -23266.808} C_VEL
LIN {X 0,Y 164.304,Z 361.018,A -85,B 0,C 180,E1 -23270.347,E2 -23270.347} C_VEL
LIN {X 0,Y 164.34,Z 361.012,A -85,B 0,C 180,E1 -23274.342,E2 -23274.342} C_VEL
LIN {X 0,Y 164.386,Z 361.008,A -85,B 0,C 180,E1 -23279.134,E2 -23279.134} C_VEL
LIN {X 0,Y 164.413,Z 361.001,A -85,B 0,C 180,E1 -23284.694,E2 -23284.694} C_VEL
LIN {X 0,Y 164.482,Z 360.996,A -85,B 0,C 180,E1 -23290.051,E2 -23290.051} C_VEL
LIN {X 0,Y 164.551,Z 360.986,A -85,B 0,C 180,E1 -23295.152,E2 -23295.152} C_VEL
LIN {X 0,Y 164.85,Z 360.948,A -85,B 0,C 180,E1 -23300.182,E2 -23300.182} C_VEL
LIN {X 0,Y 164.774,Z 360.959,A -85,B 0,C 180,E1 -23305.107,E2 -23305.107} C_VEL
LIN {X 0,Y 165.294,Z 360.89,A -85,B 0,C 180,E1 -23310,E2 -23310} C_VEL
LIN {X 0,Y 164.774,Z 360.959,A -85,B 0,C 180,E1 -23314.894,E2 -23314.894} C_VEL
LIN {X 0,Y 164.86,Z 360.945,A -85,B 0,C 180,E1 -23317.348,E2 -23317.348} C_VEL
LIN {X 0,Y 164.778,Z 360.958,A -85,B 0,C 180,E1 -23321.198,E2 -23321.198} C_VEL
LIN {X 0,Y 164.503,Z 360.987,A -85,B 0,C 180,E1 -23327.402,E2 -23327.402} C_VEL
LIN {X 0,Y 164.472,Z 360.997,A -85,B 0,C 180,E1 -23329.99,E2 -23329.99} C_VEL
LIN {X 0,Y 164.391,Z 361.003,A -85,B 0,C 180,E1 -23336.135,E2 -23336.135} C_VEL
LIN {X 0,Y 164.373,Z 361.008,A -85,B 0,C 180,E1 -23341.228,E2 -23341.228} C_VEL
LIN {X 0,Y 164.312,Z 361.016,A -85,B 0,C 180,E1 -23346.786,E2 -23346.786} C_VEL
LIN {X 0,Y 164.299,Z 361.02,A -85,B 0,C 180,E1 -23349.915,E2 -23349.915} C_VEL
LIN {X 0,Y 164.278,Z 361.016,A -85,B 0,C 180,E1 -23353.343,E2 -23353.343} C_VEL
LIN {X 0,Y 164.292,Z 361.019,A -85,B 0,C 180,E1 -23356.81,E2 -23356.81} C_VEL
LIN {X 0,Y 164.422,Z 361.001,A -85,B 0,C 180,E1 -23362.58,E2 -23362.58} C_VEL
LIN {X 0,Y 172.351,Z 389.348,A -85,B 0,C 180,E1 -23365.049,E2 -23365.049} C_VEL
LIN {X 0,Y 169.745,Z 448.767,A -85,B 0,C 180,E1 -23369.266,E2 -23369.266} C_VEL
LIN {X 0,Y 168.829,Z 463.242,A -85,B 0,C 180,E1 -23370.817,E2 -23370.817} C_VEL
LIN {X 0,Y 167.86,Z 475.59,A -85,B 0,C 180,E1 -23372.579,E2 -23372.579} C_VEL
LIN {X 0,Y 166.636,Z 489.036,A -85,B 0,C 180,E1 -23375.056,E2 -23375.056} C_VEL
LIN {X 0,Y 165.513,Z 501.069,A -85,B 0,C 180,E1 -23377.862,E2 -23377.862} C_VEL
LIN {X 0,Y 164.659,Z 510.975,A -85,B 0,C 180,E1 -23380.685,E2 -23380.685} C_VEL
LIN {X 0,Y 164.011,Z 520.07,A -85,B 0,C 180,E1 -23383.829,E2 -23383.829} C_VEL
LIN {X 0,Y 163.539,Z 528.984,A -85,B 0,C 180,E1 -23387.593,E2 -23387.593} C_VEL
LIN {X 0,Y 163.699,Z 536.642,A -85,B 0,C 180,E1 -23391.519,E2 -23391.519} C_VEL
LIN {X 0,Y 164.187,Z 542.308,A -85,B 0,C 180,E1 -23395.09,E2 -23395.09} C_VEL
LIN {X 0,Y 165.269,Z 547.101,A -85,B 0,C 180,E1 -23398.783,E2 -23398.783} C_VEL
LIN {X 0,Y 167.086,Z 550.89,A -85,B 0,C 180,E1 -23402.412,E2 -23402.412} C_VEL
LIN {X 0,Y 169.665,Z 553.886,A -85,B 0,C 180,E1 -23406.195,E2 -23406.195} C_VEL
LIN {X 0,Y 172.518,Z 555.645,A -85,B 0,C 180,E1 -23409.379,E2 -23409.379} C_VEL
LIN {X 0,Y 174.922,Z 556.469,A -85,B 0,C 180,E1 -23411.59,E2 -23411.59} C_VEL
LIN {X 0,Y 177.597,Z 556.889,A -85,B 0,C 180,E1 -23413.736,E2 -23413.736} C_VEL
LIN {X 0,Y 183.702,Z 556.544,A -85,B 0,C 180,E1 -23417.823,E2 -23417.823} C_VEL
LIN {X 0,Y 187.048,Z 555.829,A -85,B 0,C 180,E1 -23419.766,E2 -23419.766} C_VEL
LIN {X 0,Y 190.697,Z 554.718,A -85,B 0,C 180,E1 -23421.627,E2 -23421.627} C_VEL
LIN {X 0,Y 194.5,Z 553.18,A -85,B 0,C 180,E1 -23423.421,E2 -23423.421} C_VEL
LIN {X 0,Y 202.778,Z 548.877,A -85,B 0,C 180,E1 -23426.781,E2 -23426.781} C_VEL
LIN {X 0,Y 210.183,Z 543.864,A -85,B 0,C 180,E1 -23429.37,E2 -23429.37} C_VEL
LIN {X 0,Y 218.907,Z 536.726,A -85,B 0,C 180,E1 -23431.988,E2 -23431.988} C_VEL
LIN {X 0,Y 226.306,Z 529.376,A -85,B 0,C 180,E1 -23433.987,E2 -23433.987} C_VEL
LIN {X 0,Y 232.81,Z 521.949,A -85,B 0,C 180,E1 -23435.558,E2 -23435.558} C_VEL
LIN {X 0,Y 241.001,Z 510.772,A -85,B 0,C 180,E1 -23437.397,E2 -23437.397} C_VEL
LIN {X 0,Y 248.091,Z 499.041,A -85,B 0,C 180,E1 -23438.813,E2 -23438.813} C_VEL
LIN {X 0,Y 251.427,Z 492.41,A -85,B 0,C 180,E1 -23439.489,E2 -23439.489} C_VEL
LIN {X 0,Y 250.785,Z 493.908,A -85,B 0,C 180,E1 -23439.813,E2 -23439.813} C_VEL
LIN {X 0,Y 244.191,Z 506.871,A -85,B 0,C 180,E1 -23440.615,E2 -23440.615} C_VEL
LIN {X 0,Y 237.116,Z 518.455,A -85,B 0,C 180,E1 -23441.547,E2 -23441.547} C_VEL
LIN {X 0,Y 228.155,Z 531.047,A -85,B 0,C 180,E1 -23442.96,E2 -23442.96} C_VEL
LIN {X 0,Y 219.582,Z 541.347,A -85,B 0,C 180,E1 -23444.525,E2 -23444.525} C_VEL
LIN {X 0,Y 211.261,Z 550.213,A -85,B 0,C 180,E1 -23446.346,E2 -23446.346} C_VEL
LIN {X 0,Y 202.291,Z 558.592,A -85,B 0,C 180,E1 -23448.692,E2 -23448.692} C_VEL
LIN {X 0,Y 195.19,Z 564.578,A -85,B 0,C 180,E1 -23450.941,E2 -23450.941} C_VEL
LIN {X 0,Y 188.156,Z 570.006,A -85,B 0,C 180,E1 -23453.712,E2 -23453.712} C_VEL
LIN {X 0,Y 184.588,Z 572.243,A -85,B 0,C 180,E1 -23454.997,E2 -23454.997} C_VEL
LIN {X 0,Y 177.389,Z 575.331,A -85,B 0,C 180,E1 -23456.934,E2 -23456.934} C_VEL
LIN {X 0,Y 170.448,Z 577.65,A -85,B 0,C 180,E1 -23459.114,E2 -23459.114} C_VEL
LIN {X 0,Y 167.365,Z 578.705,A -85,B 0,C 180,E1 -23460.765,E2 -23460.765} C_VEL
LIN {X 0,Y 162.247,Z 580.697,A -85,B 0,C 180,E1 -23465.46,E2 -23465.46} C_VEL
LIN {X 0,Y 159.444,Z 581.338,A -85,B 0,C 180,E1 -23469.351,E2 -23469.351} C_VEL
LIN {X 0,Y 157.308,Z 581.006,A -85,B 0,C 180,E1 -23474.451,E2 -23474.451} C_VEL
LIN {X 0,Y 156.921,Z 579.168,A -85,B 0,C 180,E1 -23480.173,E2 -23480.173} C_VEL
LIN {X 0,Y 158.064,Z 576.42,A -85,B 0,C 180,E1 -23484.898,E2 -23484.898} C_VEL
LIN {X 0,Y 159.58,Z 573.073,A -85,B 0,C 180,E1 -23488.738,E2 -23488.738} C_VEL
LIN {X 0,Y 160.603,Z 570.158,A -85,B 0,C 180,E1 -23491.41,E2 -23491.41} C_VEL
LIN {X 0,Y 159.013,Z 573.78,A -85,B 0,C 180,E1 -23495.071,E2 -23495.071} C_VEL
LIN {X 0,Y 157.649,Z 577.304,A -85,B 0,C 180,E1 -23500.272,E2 -23500.272} C_VEL
LIN {X 0,Y 157.799,Z 579.46,A -85,B 0,C 180,E1 -23505.499,E2 -23505.499} C_VEL
LIN {X 0,Y 159.703,Z 580.45,A -85,B 0,C 180,E1 -23510.613,E2 -23510.613} C_VEL
LIN {X 0,Y 163.295,Z 580.308,A -85,B 0,C 180,E1 -23515.492,E2 -23515.492} C_VEL
LIN {X 0,Y 168.555,Z 579.053,A -85,B 0,C 180,E1 -23520.023,E2 -23520.023} C_VEL
LIN {X 0,Y 175.248,Z 576.652,A -85,B 0,C 180,E1 -23524.156,E2 -23524.156} C_VEL
LIN {X 0,Y 183.23,Z 573.063,A -85,B 0,C 180,E1 -23527.857,E2 -23527.857} C_VEL
LIN {X 0,Y 192.326,Z 568.224,A -85,B 0,C 180,E1 -23531.129,E2 -23531.129} C_VEL
LIN {X 0,Y 202.391,Z 562.013,A -85,B 0,C 180,E1 -23533.987,E2 -23533.987} C_VEL
LIN {X 0,Y 211.957,Z 555.266,A -85,B 0,C 180,E1 -23536.152,E2 -23536.152} C_VEL
LIN {X 0,Y 222.182,Z 547.08,A -85,B 0,C 180,E1 -23538.017,E2 -23538.017} C_VEL
LIN {X 0,Y 226.16,Z 543.621,A -85,B 0,C 180,E1 -23538.645,E2 -23538.645} C_VEL
LIN {X 0,Y 225.805,Z 543.651,A -85,B 0,C 180,E1 -23539.185,E2 -23539.185} C_VEL
LIN {X 0,Y 217.831,Z 548.895,A -85,B 0,C 180,E1 -23540.999,E2 -23540.999} C_VEL
LIN {X 0,Y 210.136,Z 553.112,A -85,B 0,C 180,E1 -23542.985,E2 -23542.985} C_VEL
LIN {X 0,Y 200.463,Z 557.248,A -85,B 0,C 180,E1 -23545.878,E2 -23545.878} C_VEL
LIN {X 0,Y 191.499,Z 559.864,A -85,B 0,C 180,E1 -23549.082,E2 -23549.082} C_VEL
LIN {X 0,Y 183.305,Z 561.015,A -85,B 0,C 180,E1 -23552.606,E2 -23552.606} C_VEL
LIN {X 0,Y 176.08,Z 560.703,A -85,B 0,C 180,E1 -23556.475,E2 -23556.475} C_VEL
LIN {X 0,Y 169.823,Z 558.991,A -85,B 0,C 180,E1 -23560.665,E2 -23560.665} C_VEL
LIN {X 0,Y 164.759,Z 555.801,A -85,B 0,C 180,E1 -23565.17,E2 -23565.17} C_VEL
LIN {X 0,Y 160.93,Z 551.099,A -85,B 0,C 180,E1 -23569.939,E2 -23569.939} C_VEL
LIN {X 0,Y 158.866,Z 546.505,A -85,B 0,C 180,E1 -23573.649,E2 -23573.649} C_VEL
LIN {X 0,Y 157.327,Z 539.874,A -85,B 0,C 180,E1 -23578.079,E2 -23578.079} C_VEL
LIN {X 0,Y 156.546,Z 531.587,A -85,B 0,C 180,E1 -23582.572,E2 -23582.572} C_VEL
LIN {X 0,Y 156.762,Z 522.994,A -85,B 0,C 180,E1 -23586.434,E2 -23586.434} C_VEL
LIN {X 0,Y 157.158,Z 513.87,A -85,B 0,C 180,E1 -23589.834,E2 -23589.834} C_VEL
LIN {X 0,Y 157.829,Z 502.961,A -85,B 0,C 180,E1 -23593.191,E2 -23593.191} C_VEL
LIN {X 0,Y 158.805,Z 490.142,A -85,B 0,C 180,E1 -23596.386,E2 -23596.386} C_VEL
LIN {X 0,Y 159.757,Z 477.234,A -85,B 0,C 180,E1 -23598.93,E2 -23598.93} C_VEL
LIN {X 0,Y 160.712,Z 464.104,A -85,B 0,C 180,E1 -23600.979,E2 -23600.979} C_VEL
LIN {X 0,Y 161.548,Z 449.071,A -85,B 0,C 180,E1 -23602.711,E2 -23602.711} C_VEL
LIN {X 0,Y 162.404,Z 426.512,A -85,B 0,C 180,E1 -23604.581,E2 -23604.581} C_VEL
LIN {X 0,Y 163.957,Z 386.984,A -85,B 0,C 180,E1 -23607.733,E2 -23607.733} C_VEL
LIN {X 0,Y 157.675,Z 363.106,A -85,B 0,C 180,E1 -23609.839,E2 -23609.839} C_VEL
LIN {X 0,Y 157.448,Z 361.866,A -85,B 0,C 180,E1 -23609.997,E2 -23609.997} C_VEL
LIN {X 0,Y 157.266,Z 361.894,A -85,B 0,C 180,E1 -23616.448,E2 -23616.448} C_VEL
LIN {X 0,Y 157.208,Z 361.901,A -85,B 0,C 180,E1 -23622.11,E2 -23622.11} C_VEL
LIN {X 0,Y 157.211,Z 361.897,A -85,B 0,C 180,E1 -23627.89,E2 -23627.89} C_VEL
LIN {X 0,Y 157.28,Z 361.891,A -85,B 0,C 180,E1 -23633.543,E2 -23633.543} C_VEL
LIN {X 0,Y 157.291,Z 361.89,A -85,B 0,C 180,E1 -23638.095,E2 -23638.095} C_VEL
LIN {X 0,Y 157.319,Z 361.883,A -85,B 0,C 180,E1 -23643.466,E2 -23643.466} C_VEL
LIN {X 0,Y 157.391,Z 361.878,A -85,B 0,C 180,E1 -23649.667,E2 -23649.667} C_VEL
LIN {X 0,Y 157.476,Z 361.867,A -85,B 0,C 180,E1 -23654.468,E2 -23654.468} C_VEL
LIN {X 0,Y 157.77,Z 361.829,A -85,B 0,C 180,E1 -23659.736,E2 -23659.736} C_VEL
LIN {X 0,Y 157.822,Z 361.821,A -85,B 0,C 180,E1 -23662.323,E2 -23662.323} C_VEL
LIN {X 0,Y 158.256,Z 361.766,A -85,B 0,C 180,E1 -23670,E2 -23670} C_VEL
LIN {X 0,Y 157.822,Z 361.822,A -85,B 0,C 180,E1 -23677.678,E2 -23677.678} C_VEL
LIN {X 0,Y 157.704,Z 361.839,A -85,B 0,C 180,E1 -23681.363,E2 -23681.363} C_VEL
LIN {X 0,Y 157.476,Z 361.866,A -85,B 0,C 180,E1 -23685.532,E2 -23685.532} C_VEL
LIN {X 0,Y 157.368,Z 361.882,A -85,B 0,C 180,E1 -23690.934,E2 -23690.934} C_VEL
LIN {X 0,Y 157.313,Z 361.887,A -85,B 0,C 180,E1 -23696.686,E2 -23696.686} C_VEL
LIN {X 0,Y 157.276,Z 361.891,A -85,B 0,C 180,E1 -23702.428,E2 -23702.428} C_VEL
LIN {X 0,Y 157.281,Z 361.893,A -85,B 0,C 180,E1 -23706.458,E2 -23706.458} C_VEL
LIN {X 0,Y 157.212,Z 361.897,A -85,B 0,C 180,E1 -23712.111,E2 -23712.111} C_VEL
LIN {X 0,Y 157.212,Z 361.903,A -85,B 0,C 180,E1 -23717.892,E2 -23717.892} C_VEL
LIN {X 0,Y 157.387,Z 361.897,A -85,B 0,C 180,E1 -23722.246,E2 -23722.246} C_VEL
LIN {X 0,Y 165.263,Z 389.966,A -85,B 0,C 180,E1 -23724.791,E2 -23724.791} C_VEL
LIN {X 0,Y 162.618,Z 449.659,A -85,B 0,C 180,E1 -23729.242,E2 -23729.242} C_VEL
LIN {X 0,Y 161.717,Z 463.357,A -85,B 0,C 180,E1 -23730.761,E2 -23730.761} C_VEL
LIN {X 0,Y 160.706,Z 476.279,A -85,B 0,C 180,E1 -23732.667,E2 -23732.667} C_VEL
LIN {X 0,Y 159.458,Z 489.699,A -85,B 0,C 180,E1 -23735.249,E2 -23735.249} C_VEL
LIN {X 0,Y 158.39,Z 500.939,A -85,B 0,C 180,E1 -23737.981,E2 -23737.981} C_VEL
LIN {X 0,Y 157.516,Z 511.514,A -85,B 0,C 180,E1 -23741.128,E2 -23741.128} C_VEL
LIN {X 0,Y 156.887,Z 520.678,A -85,B 0,C 180,E1 -23744.41,E2 -23744.41} C_VEL
LIN {X 0,Y 156.496,Z 529.686,A -85,B 0,C 180,E1 -23748.342,E2 -23748.342} C_VEL
LIN {X 0,Y 156.777,Z 538.128,A -85,B 0,C 180,E1 -23752.92,E2 -23752.92} C_VEL
LIN {X 0,Y 157.677,Z 544.759,A -85,B 0,C 180,E1 -23757.447,E2 -23757.447} C_VEL
LIN {X 0,Y 159.233,Z 549.281,A -85,B 0,C 180,E1 -23761.266,E2 -23761.266} C_VEL
LIN {X 0,Y 161.492,Z 552.811,A -85,B 0,C 180,E1 -23764.994,E2 -23764.994} C_VEL
LIN {X 0,Y 165.478,Z 556.126,A -85,B 0,C 180,E1 -23769.782,E2 -23769.782} C_VEL
LIN {X 0,Y 167.934,Z 557.2,A -85,B 0,C 180,E1 -23772.079,E2 -23772.079} C_VEL
LIN {X 0,Y 173.74,Z 558.149,A -85,B 0,C 180,E1 -23776.45,E2 -23776.45} C_VEL
LIN {X 0,Y 180.495,Z 557.645,A -85,B 0,C 180,E1 -23780.515,E2 -23780.515} C_VEL
LIN {X 0,Y 188.207,Z 555.539,A -85,B 0,C 180,E1 -23784.254,E2 -23784.254} C_VEL
LIN {X 0,Y 194.545,Z 552.945,A -85,B 0,C 180,E1 -23786.845,E2 -23786.845} C_VEL
LIN {X 0,Y 201.64,Z 549.159,A -85,B 0,C 180,E1 -23789.382,E2 -23789.382} C_VEL
LIN {X 0,Y 208.431,Z 544.775,A -85,B 0,C 180,E1 -23791.51,E2 -23791.51} C_VEL
LIN {X 0,Y 217.222,Z 537.927,A -85,B 0,C 180,E1 -23793.926,E2 -23793.926} C_VEL
LIN {X 0,Y 225.171,Z 530.465,A -85,B 0,C 180,E1 -23795.875,E2 -23795.875} C_VEL
LIN {X 0,Y 233.487,Z 521.232,A -85,B 0,C 180,E1 -23797.691,E2 -23797.691} C_VEL
LIN {X 0,Y 239.99,Z 512.662,A -85,B 0,C 180,E1 -23799.023,E2 -23799.023} C_VEL
LIN {X 0,Y 238.939,Z 514.353,A -85,B 0,C 180,E1 -23799.456,E2 -23799.456} C_VEL
LIN {X 0,Y 231.106,Z 525.458,A -85,B 0,C 180,E1 -23800.512,E2 -23800.512} C_VEL
LIN {X 0,Y 222.275,Z 536.173,A -85,B 0,C 180,E1 -23801.861,E2 -23801.861} C_VEL
LIN {X 0,Y 213.216,Z 545.767,A -85,B 0,C 180,E1 -23803.517,E2 -23803.517} C_VEL
LIN {X 0,Y 203.562,Z 554.682,A -85,B 0,C 180,E1 -23805.642,E2 -23805.642} C_VEL
LIN {X 0,Y 194.568,Z 561.991,A -85,B 0,C 180,E1 -23808.068,E2 -23808.068} C_VEL
LIN {X 0,Y 185.258,Z 568.635,A -85,B 0,C 180,E1 -23811.247,E2 -23811.247} C_VEL
LIN {X 0,Y 177.072,Z 573.773,A -85,B 0,C 180,E1 -23814.864,E2 -23814.864} C_VEL
LIN {X 0,Y 171.646,Z 576.697,A -85,B 0,C 180,E1 -23817.84,E2 -23817.84} C_VEL
LIN {X 0,Y 167.365,Z 578.705,A -85,B 0,C 180,E1 -23820.765,E2 -23820.765} C_VEL
LIN {X 0,Y 164.508,Z 579.647,A -85,B 0,C 180,E1 -23822.528,E2 -23822.528} C_VEL
LIN {X 0,Y 158.705,Z 580.299,A -85,B 0,C 180,E1 -23825.369,E2 -23825.369} C_VEL
LIN {X 0,Y 153.532,Z 580.161,A -85,B 0,C 180,E1 -23828.456,E2 -23828.456} C_VEL
LIN {X 0,Y 151.728,Z 579.87,A -85,B 0,C 180,E1 -23830.557,E2 -23830.557} C_VEL
LIN {X 0,Y 150.133,Z 578.6,A -85,B 0,C 180,E1 -23836.463,E2 -23836.463} C_VEL
LIN {X 0,Y 150.509,Z 576.034,A -85,B 0,C 180,E1 -23841.947,E2 -23841.947} C_VEL
LIN {X 0,Y 151.744,Z 573.154,A -85,B 0,C 180,E1 -23846.016,E2 -23846.016} C_VEL
LIN {X 0,Y 153.538,Z 569.2,A -85,B 0,C 180,E1 -23850,E2 -23850} C_VEL
LIN {X 0,Y 154.053,Z 567.424,A -85,B 0,C 180,E1 -23851.552,E2 -23851.552} C_VEL
LIN {X 0,Y 152.401,Z 571.147,A -85,B 0,C 180,E1 -23855.292,E2 -23855.292} C_VEL
LIN {X 0,Y 150.991,Z 574.973,A -85,B 0,C 180,E1 -23860.73,E2 -23860.73} C_VEL
LIN {X 0,Y 151.167,Z 577.444,A -85,B 0,C 180,E1 -23866.197,E2 -23866.197} C_VEL
LIN {X 0,Y 153.202,Z 578.762,A -85,B 0,C 180,E1 -23871.53,E2 -23871.53} C_VEL
LIN {X 0,Y 157.001,Z 578.984,A -85,B 0,C 180,E1 -23876.592,E2 -23876.592} C_VEL
LIN {X 0,Y 162.495,Z 578.132,A -85,B 0,C 180,E1 -23881.265,E2 -23881.265} C_VEL
LIN {X 0,Y 169.426,Z 576.17,A -85,B 0,C 180,E1 -23885.502,E2 -23885.502} C_VEL
LIN {X 0,Y 177.69,Z 573.078,A -85,B 0,C 180,E1 -23889.259,E2 -23889.259} C_VEL
LIN {X 0,Y 187.049,Z 568.791,A -85,B 0,C 180,E1 -23892.556,E2 -23892.556} C_VEL
LIN {X 0,Y 197.373,Z 563.216,A -85,B 0,C 180,E1 -23895.41,E2 -23895.41} C_VEL
LIN {X 0,Y 208.591,Z 556.131,A -85,B 0,C 180,E1 -23897.837,E2 -23897.837} C_VEL
LIN {X 0,Y 214.525,Z 551.966,A -85,B 0,C 180,E1 -23898.894,E2 -23898.894} C_VEL
LIN {X 0,Y 215.508,Z 551.135,A -85,B 0,C 180,E1 -23899.289,E2 -23899.289} C_VEL
LIN {X 0,Y 207.222,Z 555.264,A -85,B 0,C 180,E1 -23901.265,E2 -23901.265} C_VEL
LIN {X 0,Y 199.84,Z 558.232,A -85,B 0,C 180,E1 -23903.282,E2 -23903.282} C_VEL
LIN {X 0,Y 190.155,Z 560.993,A -85,B 0,C 180,E1 -23906.33,E2 -23906.33} C_VEL
LIN {X 0,Y 181.289,Z 562.317,A -85,B 0,C 180,E1 -23909.736,E2 -23909.736} C_VEL
LIN {X 0,Y 177.137,Z 562.465,A -85,B 0,C 180,E1 -23911.567,E2 -23911.567} C_VEL
LIN {X 0,Y 169.634,Z 561.642,A -85,B 0,C 180,E1 -23915.523,E2 -23915.523} C_VEL
LIN {X 0,Y 163.158,Z 559.416,A -85,B 0,C 180,E1 -23919.842,E2 -23919.842} C_VEL
LIN {X 0,Y 157.912,Z 555.775,A -85,B 0,C 180,E1 -23924.511,E2 -23924.511} C_VEL
LIN {X 0,Y 153.944,Z 550.574,A -85,B 0,C 180,E1 -23929.477,E2 -23929.477} C_VEL
LIN {X 0,Y 151.278,Z 543.753,A -85,B 0,C 180,E1 -23934.667,E2 -23934.667} C_VEL
LIN {X 0,Y 149.949,Z 536.166,A -85,B 0,C 180,E1 -23939.327,E2 -23939.327} C_VEL
LIN {X 0,Y 149.652,Z 526.877,A -85,B 0,C 180,E1 -23944.038,E2 -23944.038} C_VEL
LIN {X 0,Y 149.842,Z 518.69,A -85,B 0,C 180,E1 -23947.473,E2 -23947.473} C_VEL
LIN {X 0,Y 150.437,Z 508.123,A -85,B 0,C 180,E1 -23951.169,E2 -23951.169} C_VEL
LIN {X 0,Y 151.189,Z 496.59,A -85,B 0,C 180,E1 -23954.468,E2 -23954.468} C_VEL
LIN {X 0,Y 152.08,Z 485.16,A -85,B 0,C 180,E1 -23957.133,E2 -23957.133} C_VEL
LIN {X 0,Y 153.138,Z 470.892,A -85,B 0,C 180,E1 -23959.782,E2 -23959.782} C_VEL
LIN {X 0,Y 154.059,Z 456.699,A -85,B 0,C 180,E1 -23961.755,E2 -23961.755} C_VEL
LIN {X 0,Y 154.911,Z 441.302,A -85,B 0,C 180,E1 -23963.299,E2 -23963.299} C_VEL
LIN {X 0,Y 156.8,Z 387.761,A -85,B 0,C 180,E1 -23967.827,E2 -23967.827} C_VEL
LIN {X 0,Y 150.742,Z 364.458,A -85,B 0,C 180,E1 -23969.969,E2 -23969.969} C_VEL
LIN {X 0,Y 150.403,Z 362.743,A -85,B 0,C 180,E1 -23970.193,E2 -23970.193} C_VEL
LIN {X 0,Y 150.194,Z 362.775,A -85,B 0,C 180,E1 -23974.159,E2 -23974.159} C_VEL
LIN {X 0,Y 150.171,Z 362.774,A -85,B 0,C 180,E1 -23977.472,E2 -23977.472} C_VEL
LIN {X 0,Y 150.148,Z 362.781,A -85,B 0,C 180,E1 -23981.504,E2 -23981.504} C_VEL
LIN {X 0,Y 150.123,Z 362.781,A -85,B 0,C 180,E1 -23985.395,E2 -23985.395} C_VEL
LIN {X 0,Y 150.154,Z 362.78,A -85,B 0,C 180,E1 -23989.06,E2 -23989.06} C_VEL
LIN {X 0,Y 150.213,Z 362.774,A -85,B 0,C 180,E1 -23992.689,E2 -23992.689} C_VEL
LIN {X 0,Y 150.215,Z 362.771,A -85,B 0,C 180,E1 -23997.366,E2 -23997.366} C_VEL
LIN {X 0,Y 150.241,Z 362.767,A -85,B 0,C 180,E1 -24002.718,E2 -24002.718} C_VEL
LIN {X 0,Y 150.348,Z 362.756,A -85,B 0,C 180,E1 -24009.207,E2 -24009.207} C_VEL
LIN {X 0,Y 150.38,Z 362.748,A -85,B 0,C 180,E1 -24013.716,E2 -24013.716} C_VEL
LIN {X 0,Y 150.686,Z 362.712,A -85,B 0,C 180,E1 -24019.248,E2 -24019.248} C_VEL
LIN {X 0,Y 150.761,Z 362.699,A -85,B 0,C 180,E1 -24021.961,E2 -24021.961} C_VEL
LIN {X 0,Y 151.216,Z 362.643,A -85,B 0,C 180,E1 -24030,E2 -24030} C_VEL
LIN {X 0,Y 150.761,Z 362.701,A -85,B 0,C 180,E1 -24038.04,E2 -24038.04} C_VEL
LIN {X 0,Y 150.633,Z 362.72,A -85,B 0,C 180,E1 -24041.547,E2 -24041.547} C_VEL
LIN {X 0,Y 150.381,Z 362.748,A -85,B 0,C 180,E1 -24046.285,E2 -24046.285} C_VEL
LIN {X 0,Y 150.349,Z 362.756,A -85,B 0,C 180,E1 -24050.794,E2 -24050.794} C_VEL
LIN {X 0,Y 150.242,Z 362.767,A -85,B 0,C 180,E1 -24057.283,E2 -24057.283} C_VEL
LIN {X 0,Y 150.216,Z 362.769,A -85,B 0,C 180,E1 -24062.635,E2 -24062.635} C_VEL
LIN {X 0,Y 150.21,Z 362.773,A -85,B 0,C 180,E1 -24067.463,E2 -24067.463} C_VEL
LIN {X 0,Y 150.153,Z 362.778,A -85,B 0,C 180,E1 -24071.508,E2 -24071.508} C_VEL
LIN {X 0,Y 150.125,Z 362.783,A -85,B 0,C 180,E1 -24075.397,E2 -24075.397} C_VEL
LIN {X 0,Y 150.335,Z 362.841,A -85,B 0,C 180,E1 -24081.881,E2 -24081.881} C_VEL
LIN {X 0,Y 158.128,Z 390.789,A -85,B 0,C 180,E1 -24084.538,E2 -24084.538} C_VEL
LIN {X 0,Y 155.567,Z 449.146,A -85,B 0,C 180,E1 -24089.094,E2 -24089.094} C_VEL
LIN {X 0,Y 154.695,Z 462.358,A -85,B 0,C 180,E1 -24090.58,E2 -24090.58} C_VEL
LIN {X 0,Y 153.544,Z 476.608,A -85,B 0,C 180,E1 -24092.762,E2 -24092.762} C_VEL
LIN {X 0,Y 152.293,Z 490.037,A -85,B 0,C 180,E1 -24095.461,E2 -24095.461} C_VEL
LIN {X 0,Y 151.211,Z 501.577,A -85,B 0,C 180,E1 -24098.369,E2 -24098.369} C_VEL
LIN {X 0,Y 150.283,Z 513.052,A -85,B 0,C 180,E1 -24101.953,E2 -24101.953} C_VEL
LIN {X 0,Y 149.751,Z 521.189,A -85,B 0,C 180,E1 -24105.043,E2 -24105.043} C_VEL
LIN {X 0,Y 149.458,Z 530.213,A -85,B 0,C 180,E1 -24109.16,E2 -24109.16} C_VEL
LIN {X 0,Y 149.85,Z 538.752,A -85,B 0,C 180,E1 -24113.944,E2 -24113.944} C_VEL
LIN {X 0,Y 150.933,Z 545.451,A -85,B 0,C 180,E1 -24118.667,E2 -24118.667} C_VEL
LIN {X 0,Y 153.496,Z 551.383,A -85,B 0,C 180,E1 -24123.939,E2 -24123.939} C_VEL
LIN {X 0,Y 156.225,Z 554.683,A -85,B 0,C 180,E1 -24127.757,E2 -24127.757} C_VEL
LIN {X 0,Y 158.418,Z 556.411,A -85,B 0,C 180,E1 -24130.223,E2 -24130.223} C_VEL
LIN {X 0,Y 163.803,Z 558.663,A -85,B 0,C 180,E1 -24134.919,E2 -24134.919} C_VEL
LIN {X 0,Y 170.334,Z 559.44,A -85,B 0,C 180,E1 -24139.275,E2 -24139.275} C_VEL
LIN {X 0,Y 177.82,Z 558.682,A -85,B 0,C 180,E1 -24143.281,E2 -24143.281} C_VEL
LIN {X 0,Y 186.231,Z 556.425,A -85,B 0,C 180,E1 -24146.928,E2 -24146.928} C_VEL
LIN {X 0,Y 194.759,Z 552.887,A -85,B 0,C 180,E1 -24149.996,E2 -24149.996} C_VEL
LIN {X 0,Y 202.81,Z 548.455,A -85,B 0,C 180,E1 -24152.489,E2 -24152.489} C_VEL
LIN {X 0,Y 210.573,Z 543.308,A -85,B 0,C 180,E1 -24154.569,E2 -24154.569} C_VEL
LIN {X 0,Y 219.778,Z 535.928,A -85,B 0,C 180,E1 -24156.784,E2 -24156.784} C_VEL
LIN {X 0,Y 228.744,Z 527.215,A -85,B 0,C 180,E1 -24158.672,E2 -24158.672} C_VEL
LIN {X 0,Y 227.894,Z 528.303,A -85,B 0,C 180,E1 -24159.01,E2 -24159.01} C_VEL
LIN {X 0,Y 218.252,Z 538.987,A -85,B 0,C 180,E1 -24160.417,E2 -24160.417} C_VEL
LIN {X 0,Y 210.063,Z 546.817,A -85,B 0,C 180,E1 -24161.819,E2 -24161.819} C_VEL
LIN {X 0,Y 199.979,Z 555.349,A -85,B 0,C 180,E1 -24163.908,E2 -24163.908} C_VEL
LIN {X 0,Y 189.385,Z 563.12,A -85,B 0,C 180,E1 -24166.643,E2 -24166.643} C_VEL
LIN {X 0,Y 182.092,Z 567.782,A -85,B 0,C 180,E1 -24168.994,E2 -24168.994} C_VEL
LIN {X 0,Y 173.418,Z 572.764,A -85,B 0,C 180,E1 -24172.562,E2 -24172.562} C_VEL
LIN {X 0,Y 165.692,Z 576.365,A -85,B 0,C 180,E1 -24176.536,E2 -24176.536} C_VEL
LIN {X 0,Y 159.359,Z 578.722,A -85,B 0,C 180,E1 -24180.979,E2 -24180.979} C_VEL
LIN {X 0,Y 154.596,Z 579.876,A -85,B 0,C 180,E1 -24185.848,E2 -24185.848} C_VEL
LIN {X 0,Y 151.728,Z 579.87,A -85,B 0,C 180,E1 -24190.557,E2 -24190.557} C_VEL
LIN {X 0,Y 150.232,Z 579.417,A -85,B 0,C 180,E1 -24192.719,E2 -24192.719} C_VEL
LIN {X 0,Y 146.772,Z 577.615,A -85,B 0,C 180,E1 -24196.235,E2 -24196.235} C_VEL
LIN {X 0,Y 144.463,Z 575.597,A -85,B 0,C 180,E1 -24199.121,E2 -24199.121} C_VEL
LIN {X 0,Y 143.801,Z 573.977,A -85,B 0,C 180,E1 -24201.368,E2 -24201.368} C_VEL
LIN {X 0,Y 143.893,Z 573.45,A -85,B 0,C 180,E1 -24202.125,E2 -24202.125} C_VEL
LIN {X 0,Y 145.668,Z 569.503,A -85,B 0,C 180,E1 -24207.234,E2 -24207.234} C_VEL
LIN {X 0,Y 146.933,Z 566.572,A -85,B 0,C 180,E1 -24210,E2 -24210} C_VEL
LIN {X 0,Y 147.55,Z 564.575,A -85,B 0,C 180,E1 -24211.705,E2 -24211.705} C_VEL
LIN {X 0,Y 145.862,Z 568.394,A -85,B 0,C 180,E1 -24215.529,E2 -24215.529} C_VEL
LIN {X 0,Y 144.378,Z 572.509,A -85,B 0,C 180,E1 -24221.227,E2 -24221.227} C_VEL
LIN {X 0,Y 144.622,Z 575.299,A -85,B 0,C 180,E1 -24226.952,E2 -24226.952} C_VEL
LIN {X 0,Y 146.779,Z 576.943,A -85,B 0,C 180,E1 -24232.522,E2 -24232.522} C_VEL
LIN {X 0,Y 150.786,Z 577.518,A -85,B 0,C 180,E1 -24237.781,E2 -24237.781} C_VEL
LIN {X 0,Y 156.519,Z 577.059,A -85,B 0,C 180,E1 -24242.603,E2 -24242.603} C_VEL
LIN {X 0,Y 163.727,Z 575.534,A -85,B 0,C 180,E1 -24246.938,E2 -24246.938} C_VEL
LIN {X 0,Y 172.266,Z 572.926,A -85,B 0,C 180,E1 -24250.75,E2 -24250.75} C_VEL
LIN {X 0,Y 181.898,Z 569.18,A -85,B 0,C 180,E1 -24254.064,E2 -24254.064} C_VEL
LIN {X 0,Y 192.485,Z 564.211,A -85,B 0,C 180,E1 -24256.906,E2 -24256.906} C_VEL
LIN {X 0,Y 203.932,Z 557.85,A -85,B 0,C 180,E1 -24259.304,E2 -24259.304} C_VEL
LIN {X 0,Y 199.714,Z 559.238,A -85,B 0,C 180,E1 -24260.695,E2 -24260.695} C_VEL
LIN {X 0,Y 189.39,Z 562.177,A -85,B 0,C 180,E1 -24263.576,E2 -24263.576} C_VEL
LIN {X 0,Y 179.811,Z 563.623,A -85,B 0,C 180,E1 -24266.824,E2 -24266.824} C_VEL
LIN {X 0,Y 171.004,Z 563.715,A -85,B 0,C 180,E1 -24270.449,E2 -24270.449} C_VEL
LIN {X 0,Y 163.219,Z 562.408,A -85,B 0,C 180,E1 -24274.494,E2 -24274.494} C_VEL
LIN {X 0,Y 156.511,Z 559.666,A -85,B 0,C 180,E1 -24278.946,E2 -24278.946} C_VEL
LIN {X 0,Y 151.072,Z 555.516,A -85,B 0,C 180,E1 -24283.791,E2 -24283.791} C_VEL
LIN {X 0,Y 147.922,Z 551.411,A -85,B 0,C 180,E1 -24287.653,E2 -24287.653} C_VEL
LIN {X 0,Y 144.825,Z 544.506,A -85,B 0,C 180,E1 -24293.03,E2 -24293.03} C_VEL
LIN {X 0,Y 143.261,Z 536.893,A -85,B 0,C 180,E1 -24297.89,E2 -24297.89} C_VEL
LIN {X 0,Y 142.659,Z 527.576,A -85,B 0,C 180,E1 -24302.822,E2 -24302.822} C_VEL
LIN {X 0,Y 142.854,Z 519.603,A -85,B 0,C 180,E1 -24306.354,E2 -24306.354} C_VEL
LIN {X 0,Y 143.379,Z 508.62,A -85,B 0,C 180,E1 -24310.395,E2 -24310.395} C_VEL
LIN {X 0,Y 144.047,Z 497.556,A -85,B 0,C 180,E1 -24313.722,E2 -24313.722} C_VEL
LIN {X 0,Y 144.92,Z 486.098,A -85,B 0,C 180,E1 -24316.552,E2 -24316.552} C_VEL
LIN {X 0,Y 145.973,Z 471.941,A -85,B 0,C 180,E1 -24319.328,E2 -24319.328} C_VEL
LIN {X 0,Y 146.901,Z 458.001,A -85,B 0,C 180,E1 -24321.393,E2 -24321.393} C_VEL
LIN {X 0,Y 147.732,Z 442.995,A -85,B 0,C 180,E1 -24323.015,E2 -24323.015} C_VEL
LIN {X 0,Y 149.752,Z 388.782,A -85,B 0,C 180,E1 -24327.872,E2 -24327.872} C_VEL
LIN {X 0,Y 143.881,Z 366.318,A -85,B 0,C 180,E1 -24330.032,E2 -24330.032} C_VEL
LIN {X 0,Y 143.344,Z 363.623,A -85,B 0,C 180,E1 -24330.35,E2 -24330.35} C_VEL
LIN {X 0,Y 143.087,Z 363.66,A -85,B 0,C 180,E1 -24336.113,E2 -24336.113} C_VEL
LIN {X 0,Y 143.059,Z 363.661,A -85,B 0,C 180,E1 -24339.689,E2 -24339.689} C_VEL
LIN {X 0,Y 143.054,Z 363.665,A -85,B 0,C 180,E1 -24343.454,E2 -24343.454} C_VEL
LIN {X 0,Y 143.065,Z 363.659,A -85,B 0,C 180,E1 -24347.463,E2 -24347.463} C_VEL
LIN {X 0,Y 143.104,Z 363.658,A -85,B 0,C 180,E1 -24351.79,E2 -24351.79} C_VEL
LIN {X 0,Y 143.182,Z 363.647,A -85,B 0,C 180,E1 -24357.322,E2 -24357.322} C_VEL
LIN {X 0,Y 143.187,Z 363.647,A -85,B 0,C 180,E1 -24362.063,E2 -24362.063} C_VEL
LIN {X 0,Y 143.274,Z 363.638,A -85,B 0,C 180,E1 -24368.745,E2 -24368.745} C_VEL
LIN {X 0,Y 143.314,Z 363.628,A -85,B 0,C 180,E1 -24372.889,E2 -24372.889} C_VEL
LIN {X 0,Y 143.6,Z 363.596,A -85,B 0,C 180,E1 -24378.711,E2 -24378.711} C_VEL
LIN {X 0,Y 143.682,Z 363.58,A -85,B 0,C 180,E1 -24381.562,E2 -24381.562} C_VEL
LIN {X 0,Y 144.175,Z 363.52,A -85,B 0,C 180,E1 -24390,E2 -24390} C_VEL
LIN {X 0,Y 143.683,Z 363.582,A -85,B 0,C 180,E1 -24398.439,E2 -24398.439} C_VEL
LIN {X 0,Y 143.569,Z 363.6,A -85,B 0,C 180,E1 -24401.758,E2 -24401.758} C_VEL
LIN {X 0,Y 143.314,Z 363.626,A -85,B 0,C 180,E1 -24407.112,E2 -24407.112} C_VEL
LIN {X 0,Y 143.275,Z 363.637,A -85,B 0,C 180,E1 -24411.256,E2 -24411.256} C_VEL
LIN {X 0,Y 143.189,Z 363.647,A -85,B 0,C 180,E1 -24417.938,E2 -24417.938} C_VEL
LIN {X 0,Y 143.167,Z 363.647,A -85,B 0,C 180,E1 -24423.436,E2 -24423.436} C_VEL
LIN {X 0,Y 143.074,Z 363.663,A -85,B 0,C 180,E1 -24429.687,E2 -24429.687} C_VEL
LIN {X 0,Y 143.056,Z 363.659,A -85,B 0,C 180,E1 -24433.456,E2 -24433.456} C_VEL
LIN {X 0,Y 143.067,Z 363.664,A -85,B 0,C 180,E1 -24437.466,E2 -24437.466} C_VEL
LIN {X 0,Y 143.266,Z 363.632,A -85,B 0,C 180,E1 -24441.505,E2 -24441.505} C_VEL
LIN {X 0,Y 151.049,Z 391.773,A -85,B 0,C 180,E1 -24444.3,E2 -24444.3} C_VEL
LIN {X 0,Y 148.428,Z 449.662,A -85,B 0,C 180,E1 -24449.108,E2 -24449.108} C_VEL
LIN {X 0,Y 147.509,Z 463.695,A -85,B 0,C 180,E1 -24450.769,E2 -24450.769} C_VEL
LIN {X 0,Y 146.432,Z 476.836,A -85,B 0,C 180,E1 -24452.875,E2 -24452.875} C_VEL
LIN {X 0,Y 145.278,Z 488.869,A -85,B 0,C 180,E1 -24455.341,E2 -24455.341} C_VEL
LIN {X 0,Y 144.25,Z 499.885,A -85,B 0,C 180,E1 -24458.158,E2 -24458.158} C_VEL
LIN {X 0,Y 143.325,Z 511.393,A -85,B 0,C 180,E1 -24461.785,E2 -24461.785} C_VEL
LIN {X 0,Y 142.654,Z 521.572,A -85,B 0,C 180,E1 -24465.741,E2 -24465.741} C_VEL
LIN {X 0,Y 142.446,Z 530.561,A -85,B 0,C 180,E1 -24469.964,E2 -24469.964} C_VEL
LIN {X 0,Y 142.853,Z 538.154,A -85,B 0,C 180,E1 -24474.355,E2 -24474.355} C_VEL
LIN {X 0,Y 143.786,Z 544.276,A -85,B 0,C 180,E1 -24478.601,E2 -24478.601} C_VEL
LIN {X 0,Y 145.572,Z 549.326,A -85,B 0,C 180,E1 -24482.769,E2 -24482.769} C_VEL
LIN {X 0,Y 149.089,Z 554.504,A -85,B 0,C 180,E1 -24488.131,E2 -24488.131} C_VEL
LIN {X 0,Y 153.968,Z 558.059,A -85,B 0,C 180,E1 -24493.194,E2 -24493.194} C_VEL
LIN {X 0,Y 160.151,Z 560.127,A -85,B 0,C 180,E1 -24497.891,E2 -24497.891} C_VEL
LIN {X 0,Y 167.377,Z 560.689,A -85,B 0,C 180,E1 -24502.205,E2 -24502.205} C_VEL
LIN {X 0,Y 175.639,Z 559.751,A -85,B 0,C 180,E1 -24506.115,E2 -24506.115} C_VEL
LIN {X 0,Y 180.102,Z 558.751,A -85,B 0,C 180,E1 -24507.923,E2 -24507.923} C_VEL
LIN {X 0,Y 188.156,Z 556.096,A -85,B 0,C 180,E1 -24510.783,E2 -24510.783} C_VEL
LIN {X 0,Y 197.174,Z 551.999,A -85,B 0,C 180,E1 -24513.538,E2 -24513.538} C_VEL
LIN {X 0,Y 205.169,Z 547.392,A -85,B 0,C 180,E1 -24515.616,E2 -24515.616} C_VEL
LIN {X 0,Y 213.567,Z 541.638,A -85,B 0,C 180,E1 -24517.565,E2 -24517.565} C_VEL
LIN {X 0,Y 216.22,Z 539.587,A -85,B 0,C 180,E1 -24518.14,E2 -24518.14} C_VEL
LIN {X 0,Y 216.01,Z 539.979,A -85,B 0,C 180,E1 -24518.66,E2 -24518.66} C_VEL
LIN {X 0,Y 207.107,Z 547.887,A -85,B 0,C 180,E1 -24520.073,E2 -24520.073} C_VEL
LIN {X 0,Y 196.577,Z 556.006,A -85,B 0,C 180,E1 -24522.11,E2 -24522.11} C_VEL
LIN {X 0,Y 186.967,Z 562.456,A -85,B 0,C 180,E1 -24524.421,E2 -24524.421} C_VEL
LIN {X 0,Y 176.819,Z 568.303,A -85,B 0,C 180,E1 -24527.491,E2 -24527.491} C_VEL
LIN {X 0,Y 167.842,Z 572.75,A -85,B 0,C 180,E1 -24531.09,E2 -24531.09} C_VEL
LIN {X 0,Y 159.834,Z 575.926,A -85,B 0,C 180,E1 -24535.136,E2 -24535.136} C_VEL
LIN {X 0,Y 153.211,Z 577.862,A -85,B 0,C 180,E1 -24539.695,E2 -24539.695} C_VEL
LIN {X 0,Y 148.19,Z 578.63,A -85,B 0,C 180,E1 -24544.733,E2 -24544.733} C_VEL
LIN {X 0,Y 144.899,Z 578.243,A -85,B 0,C 180,E1 -24550.152,E2 -24550.152} C_VEL
LIN {X 0,Y 143.412,Z 576.661,A -85,B 0,C 180,E1 -24555.816,E2 -24555.816} C_VEL
LIN {X 0,Y 143.763,Z 573.83,A -85,B 0,C 180,E1 -24561.566,E2 -24561.566} C_VEL
LIN {X 0,Y 143.893,Z 573.45,A -85,B 0,C 180,E1 -24562.125,E2 -24562.125} C_VEL
LIN {X 0,Y 143.687,Z 572.224,A -85,B 0,C 180,E1 -24563.608,E2 -24563.608} C_VEL
LIN {X 0,Y 141.894,Z 569.348,A -85,B 0,C 180,E1 -24565.919,E2 -24565.919} C_VEL
LIN {X 0,Y 140.217,Z 566.009,A -85,B 0,C 180,E1 -24568.242,E2 -24568.242} C_VEL
LIN {X 0,Y 140.262,Z 564.131,A -85,B 0,C 180,E1 -24569.713,E2 -24569.713} C_VEL
LIN {X 0,Y 141.135,Z 561.553,A -85,B 0,C 180,E1 -24571.873,E2 -24571.873} C_VEL
LIN {X 0,Y 139.378,Z 565.502,A -85,B 0,C 180,E1 -24575.788,E2 -24575.788} C_VEL
LIN {X 0,Y 137.843,Z 569.904,A -85,B 0,C 180,E1 -24581.767,E2 -24581.767} C_VEL
LIN {X 0,Y 138.157,Z 572.984,A -85,B 0,C 180,E1 -24587.771,E2 -24587.771} C_VEL
LIN {X 0,Y 140.452,Z 574.952,A -85,B 0,C 180,E1 -24593.597,E2 -24593.597} C_VEL
LIN {X 0,Y 144.666,Z 575.883,A -85,B 0,C 180,E1 -24599.065,E2 -24599.065} C_VEL
LIN {X 0,Y 150.656,Z 575.815,A -85,B 0,C 180,E1 -24604.041,E2 -24604.041} C_VEL
LIN {X 0,Y 158.154,Z 574.727,A -85,B 0,C 180,E1 -24608.471,E2 -24608.471} C_VEL
LIN {X 0,Y 166.969,Z 572.591,A -85,B 0,C 180,E1 -24612.335,E2 -24612.335} C_VEL
LIN {X 0,Y 176.883,Z 569.372,A -85,B 0,C 180,E1 -24615.658,E2 -24615.658} C_VEL
LIN {X 0,Y 187.712,Z 564.992,A -85,B 0,C 180,E1 -24618.487,E2 -24618.487} C_VEL
LIN {X 0,Y 191.591,Z 563.208,A -85,B 0,C 180,E1 -24619.344,E2 -24619.344} C_VEL
LIN {X 0,Y 192.205,Z 562.646,A -85,B 0,C 180,E1 -24620.039,E2 -24620.039} C_VEL
LIN {X 0,Y 183.911,Z 564.362,A -85,B 0,C 180,E1 -24622.306,E2 -24622.306} C_VEL
LIN {X 0,Y 174.034,Z 565.237,A -85,B 0,C 180,E1 -24625.571,E2 -24625.571} C_VEL
LIN {X 0,Y 164.919,Z 564.78,A -85,B 0,C 180,E1 -24629.243,E2 -24629.243} C_VEL
LIN {X 0,Y 156.845,Z 562.955,A -85,B 0,C 180,E1 -24633.378,E2 -24633.378} C_VEL
LIN {X 0,Y 149.893,Z 559.719,A -85,B 0,C 180,E1 -24637.969,E2 -24637.969} C_VEL
LIN {X 0,Y 144.266,Z 555.058,A -85,B 0,C 180,E1 -24643.003,E2 -24643.003} C_VEL
LIN {X 0,Y 140.073,Z 548.902,A -85,B 0,C 180,E1 -24648.421,E2 -24648.421} C_VEL
LIN {X 0,Y 137.355,Z 540.986,A -85,B 0,C 180,E1 -24654.125,E2 -24654.125} C_VEL
LIN {X 0,Y 135.988,Z 532.397,A -85,B 0,C 180,E1 -24659.258,E2 -24659.258} C_VEL
LIN {X 0,Y 135.84,Z 523.533,A -85,B 0,C 180,E1 -24663.707,E2 -24663.707} C_VEL
LIN {X 0,Y 136.15,Z 512.803,A -85,B 0,C 180,E1 -24668.159,E2 -24668.159} C_VEL
LIN {X 0,Y 136.757,Z 501.857,A -85,B 0,C 180,E1 -24671.861,E2 -24671.861} C_VEL
LIN {X 0,Y 137.723,Z 488.449,A -85,B 0,C 180,E1 -24675.538,E2 -24675.538} C_VEL
LIN {X 0,Y 138.689,Z 474.701,A -85,B 0,C 180,E1 -24678.463,E2 -24678.463} C_VEL
LIN {X 0,Y 139.609,Z 461.652,A -85,B 0,C 180,E1 -24680.632,E2 -24680.632} C_VEL
LIN {X 0,Y 140.448,Z 446.032,A -85,B 0,C 180,E1 -24682.525,E2 -24682.525} C_VEL
LIN {X 0,Y 141.415,Z 417.443,A -85,B 0,C 180,E1 -24685.281,E2 -24685.281} C_VEL
LIN {X 0,Y 142.552,Z 389.51,A -85,B 0,C 180,E1 -24687.915,E2 -24687.915} C_VEL
LIN {X 0,Y 136.819,Z 367.19,A -85,B 0,C 180,E1 -24690.149,E2 -24690.149} C_VEL
LIN {X 0,Y 136.291,Z 364.501,A -85,B 0,C 180,E1 -24690.478,E2 -24690.478} C_VEL
LIN {X 0,Y 136.066,Z 364.537,A -85,B 0,C 180,E1 -24694.621,E2 -24694.621} C_VEL
LIN {X 0,Y 136.029,Z 364.536,A -85,B 0,C 180,E1 -24699.197,E2 -24699.197} C_VEL
LIN {X 0,Y 135.995,Z 364.544,A -85,B 0,C 180,E1 -24703.657,E2 -24703.657} C_VEL
LIN {X 0,Y 136.029,Z 364.535,A -85,B 0,C 180,E1 -24707.806,E2 -24707.806} C_VEL
LIN {X 0,Y 136.053,Z 364.537,A -85,B 0,C 180,E1 -24711.693,E2 -24711.693} C_VEL
LIN {X 0,Y 136.087,Z 364.526,A -85,B 0,C 180,E1 -24715.717,E2 -24715.717} C_VEL
LIN {X 0,Y 136.143,Z 364.524,A -85,B 0,C 180,E1 -24722.316,E2 -24722.316} C_VEL
LIN {X 0,Y 136.241,Z 364.514,A -85,B 0,C 180,E1 -24728.833,E2 -24728.833} C_VEL
LIN {X 0,Y 136.283,Z 364.508,A -85,B 0,C 180,E1 -24735.058,E2 -24735.058} C_VEL
LIN {X 0,Y 136.499,Z 364.482,A -85,B 0,C 180,E1 -24738.115,E2 -24738.115} C_VEL
LIN {X 0,Y 136.606,Z 364.462,A -85,B 0,C 180,E1 -24741.122,E2 -24741.122} C_VEL
LIN {X 0,Y 137.132,Z 364.397,A -85,B 0,C 180,E1 -24750,E2 -24750} C_VEL
LIN {X 0,Y 136.607,Z 364.464,A -85,B 0,C 180,E1 -24758.879,E2 -24758.879} C_VEL
LIN {X 0,Y 136.491,Z 364.483,A -85,B 0,C 180,E1 -24761.959,E2 -24761.959} C_VEL
LIN {X 0,Y 136.25,Z 364.508,A -85,B 0,C 180,E1 -24768.029,E2 -24768.029} C_VEL
LIN {X 0,Y 136.196,Z 364.52,A -85,B 0,C 180,E1 -24771.75,E2 -24771.75} C_VEL
LIN {X 0,Y 136.114,Z 364.53,A -85,B 0,C 180,E1 -24778.629,E2 -24778.629} C_VEL
LIN {X 0,Y 136.077,Z 364.53,A -85,B 0,C 180,E1 -24784.62,E2 -24784.62} C_VEL
LIN {X 0,Y 136.049,Z 364.537,A -85,B 0,C 180,E1 -24789.21,E2 -24789.21} C_VEL
LIN {X 0,Y 135.998,Z 364.539,A -85,B 0,C 180,E1 -24793.659,E2 -24793.659} C_VEL
LIN {X 0,Y 136.175,Z 364.515,A -85,B 0,C 180,E1 -24800.729,E2 -24800.729} C_VEL
LIN {X 0,Y 136.198,Z 364.512,A -85,B 0,C 180,E1 -24801.122,E2 -24801.122} C_VEL
LIN {X 0,Y 143.958,Z 393.248,A -85,B 0,C 180,E1 -24804.14,E2 -24804.14} C_VEL
LIN {X 0,Y 141.237,Z 451.213,A -85,B 0,C 180,E1 -24809.231,E2 -24809.231} C_VEL
LIN {X 0,Y 140.309,Z 464.965,A -85,B 0,C 180,E1 -24810.973,E2 -24810.973} C_VEL
LIN {X 0,Y 139.119,Z 478.787,A -85,B 0,C 180,E1 -24813.364,E2 -24813.364} C_VEL
LIN {X 0,Y 137.875,Z 491.905,A -85,B 0,C 180,E1 -24816.327,E2 -24816.327} C_VEL
LIN {X 0,Y 136.802,Z 503.853,A -85,B 0,C 180,E1 -24819.712,E2 -24819.712} C_VEL
LIN {X 0,Y 136.015,Z 514.673,A -85,B 0,C 180,E1 -24823.491,E2 -24823.491} C_VEL
LIN {X 0,Y 135.537,Z 523.587,A -85,B 0,C 180,E1 -24827.27,E2 -24827.27} C_VEL
LIN {X 0,Y 135.524,Z 532.414,A -85,B 0,C 180,E1 -24831.803,E2 -24831.803} C_VEL
LIN {X 0,Y 136.296,Z 540.829,A -85,B 0,C 180,E1 -24837.046,E2 -24837.046} C_VEL
LIN {X 0,Y 137.742,Z 546.646,A -85,B 0,C 180,E1 -24841.463,E2 -24841.463} C_VEL
LIN {X 0,Y 140.053,Z 551.434,A -85,B 0,C 180,E1 -24845.761,E2 -24845.761} C_VEL
LIN {X 0,Y 142.262,Z 554.384,A -85,B 0,C 180,E1 -24848.867,E2 -24848.867} C_VEL
LIN {X 0,Y 146.995,Z 558.184,A -85,B 0,C 180,E1 -24853.832,E2 -24853.832} C_VEL
LIN {X 0,Y 153.355,Z 560.817,A -85,B 0,C 180,E1 -24858.712,E2 -24858.712} C_VEL
LIN {X 0,Y 160.818,Z 561.922,A -85,B 0,C 180,E1 -24863.162,E2 -24863.162} C_VEL
LIN {X 0,Y 169.367,Z 561.584,A -85,B 0,C 180,E1 -24867.16,E2 -24867.16} C_VEL
LIN {X 0,Y 173.969,Z 560.876,A -85,B 0,C 180,E1 -24868.999,E2 -24868.999} C_VEL
LIN {X 0,Y 183.777,Z 558.258,A -85,B 0,C 180,E1 -24872.371,E2 -24872.371} C_VEL
LIN {X 0,Y 191.577,Z 555.268,A -85,B 0,C 180,E1 -24874.655,E2 -24874.655} C_VEL
LIN {X 0,Y 199.788,Z 551.288,A -85,B 0,C 180,E1 -24876.729,E2 -24876.729} C_VEL
LIN {X 0,Y 205.468,Z 548.017,A -85,B 0,C 180,E1 -24878.003,E2 -24878.003} C_VEL
LIN {X 0,Y 205.423,Z 548.089,A -85,B 0,C 180,E1 -24878.104,E2 -24878.104} C_VEL
LIN {X 0,Y 193.377,Z 556.662,A -85,B 0,C 180,E1 -24880.251,E2 -24880.251} C_VEL
LIN {X 0,Y 182.102,Z 563.42,A -85,B 0,C 180,E1 -24882.837,E2 -24882.837} C_VEL
LIN {X 0,Y 171.659,Z 568.669,A -85,B 0,C 180,E1 -24885.892,E2 -24885.892} C_VEL
LIN {X 0,Y 162.39,Z 572.609,A -85,B 0,C 180,E1 -24889.519,E2 -24889.519} C_VEL
LIN {X 0,Y 154.082,Z 575.324,A -85,B 0,C 180,E1 -24893.632,E2 -24893.632} C_VEL
LIN {X 0,Y 147.153,Z 576.864,A -85,B 0,C 180,E1 -24898.307,E2 -24898.307} C_VEL
LIN {X 0,Y 141.865,Z 577.263,A -85,B 0,C 180,E1 -24903.521,E2 -24903.521} C_VEL
LIN {X 0,Y 138.383,Z 576.539,A -85,B 0,C 180,E1 -24909.175,E2 -24909.175} C_VEL
LIN {X 0,Y 136.758,Z 574.651,A -85,B 0,C 180,E1 -24915.11,E2 -24915.11} C_VEL
LIN {X 0,Y 137.087,Z 571.499,A -85,B 0,C 180,E1 -24921.152,E2 -24921.152} C_VEL
LIN {X 0,Y 138.446,Z 568.188,A -85,B 0,C 180,E1 -24925.632,E2 -24925.632} C_VEL
LIN {X 0,Y 140.262,Z 564.131,A -85,B 0,C 180,E1 -24929.713,E2 -24929.713} C_VEL
LIN {X 0,Y 140.313,Z 563.142,A -85,B 0,C 180,E1 -24931.179,E2 -24931.179} C_VEL
LIN {X 0,Y 139.527,Z 562.983,A -85,B 0,C 180,E1 -24932.695,E2 -24932.695} C_VEL
LIN {X 0,Y 138.208,Z 563.359,A -85,B 0,C 180,E1 -24934.23,E2 -24934.23} C_VEL
LIN {X 0,Y 133.216,Z 565.418,A -85,B 0,C 180,E1 -24938.97,E2 -24938.97} C_VEL
LIN {X 0,Y 131.6,Z 566.672,A -85,B 0,C 180,E1 -24941.549,E2 -24941.549} C_VEL
LIN {X 0,Y 131.412,Z 567.162,A -85,B 0,C 180,E1 -24942.435,E2 -24942.435} C_VEL
LIN {X 0,Y 131.774,Z 570.488,A -85,B 0,C 180,E1 -24948.663,E2 -24948.663} C_VEL
LIN {X 0,Y 134.233,Z 572.778,A -85,B 0,C 180,E1 -24954.762,E2 -24954.762} C_VEL
LIN {X 0,Y 138.927,Z 574.096,A -85,B 0,C 180,E1 -24960.682,E2 -24960.682} C_VEL
LIN {X 0,Y 144.924,Z 574.375,A -85,B 0,C 180,E1 -24965.586,E2 -24965.586} C_VEL
LIN {X 0,Y 152.718,Z 573.72,A -85,B 0,C 180,E1 -24970.111,E2 -24970.111} C_VEL
LIN {X 0,Y 161.811,Z 572.057,A -85,B 0,C 180,E1 -24974.022,E2 -24974.022} C_VEL
LIN {X 0,Y 172.002,Z 569.355,A -85,B 0,C 180,E1 -24977.348,E2 -24977.348} C_VEL
LIN {X 0,Y 180.611,Z 566.449,A -85,B 0,C 180,E1 -24979.597,E2 -24979.597} C_VEL
LIN {X 0,Y 181.12,Z 566.022,A -85,B 0,C 180,E1 -24980.219,E2 -24980.219} C_VEL
LIN {X 0,Y 173.294,Z 566.673,A -85,B 0,C 180,E1 -24982.53,E2 -24982.53} C_VEL
LIN {X 0,Y 163.46,Z 566.32,A -85,B 0,C 180,E1 -24986.016,E2 -24986.016} C_VEL
LIN {X 0,Y 154.602,Z 564.627,A -85,B 0,C 180,E1 -24989.996,E2 -24989.996} C_VEL
LIN {X 0,Y 146.777,Z 561.598,A -85,B 0,C 180,E1 -24994.471,E2 -24994.471} C_VEL
LIN {X 0,Y 140.242,Z 557.151,A -85,B 0,C 180,E1 -24999.463,E2 -24999.463} C_VEL
LIN {X 0,Y 135.199,Z 551.238,A -85,B 0,C 180,E1 -25004.934,E2 -25004.934} C_VEL
LIN {X 0,Y 131.936,Z 544.732,A -85,B 0,C 180,E1 -25010.029,E2 -25010.029} C_VEL
LIN {X 0,Y 129.918,Z 536.808,A -85,B 0,C 180,E1 -25015.344,E2 -25015.344} C_VEL
LIN {X 0,Y 128.929,Z 527.103,A -85,B 0,C 180,E1 -25020.779,E2 -25020.779} C_VEL
LIN {X 0,Y 129.038,Z 518.913,A -85,B 0,C 180,E1 -25024.685,E2 -25024.685} C_VEL
LIN {X 0,Y 129.431,Z 508.107,A -85,B 0,C 180,E1 -25028.98,E2 -25028.98} C_VEL
LIN {X 0,Y 130.091,Z 496.018,A -85,B 0,C 180,E1 -25032.875,E2 -25032.875} C_VEL
LIN {X 0,Y 130.937,Z 484.221,A -85,B 0,C 180,E1 -25035.965,E2 -25035.965} C_VEL
LIN {X 0,Y 132.031,Z 469.276,A -85,B 0,C 180,E1 -25039.027,E2 -25039.027} C_VEL
LIN {X 0,Y 132.846,Z 455.582,A -85,B 0,C 180,E1 -25041.123,E2 -25041.123} C_VEL
LIN {X 0,Y 133.876,Z 433.979,A -85,B 0,C 180,E1 -25043.492,E2 -25043.492} C_VEL
LIN {X 0,Y 135.418,Z 390.271,A -85,B 0,C 180,E1 -25047.92,E2 -25047.92} C_VEL
LIN {X 0,Y 129.89,Z 368.701,A -85,B 0,C 180,E1 -25050.166,E2 -25050.166} C_VEL
LIN {X 0,Y 129.255,Z 365.378,A -85,B 0,C 180,E1 -25050.595,E2 -25050.595} C_VEL
LIN {X 0,Y 128.933,Z 365.421,A -85,B 0,C 180,E1 -25056.839,E2 -25056.839} C_VEL
LIN {X 0,Y 128.932,Z 365.423,A -85,B 0,C 180,E1 -25060.85,E2 -25060.85} C_VEL
LIN {X 0,Y 128.919,Z 365.423,A -85,B 0,C 180,E1 -25065.126,E2 -25065.126} C_VEL
LIN {X 0,Y 128.955,Z 365.42,A -85,B 0,C 180,E1 -25069.727,E2 -25069.727} C_VEL
LIN {X 0,Y 128.989,Z 365.411,A -85,B 0,C 180,E1 -25074.81,E2 -25074.81} C_VEL
LIN {X 0,Y 129.031,Z 365.413,A -85,B 0,C 180,E1 -25080.646,E2 -25080.646} C_VEL
LIN {X 0,Y 129.106,Z 365.402,A -85,B 0,C 180,E1 -25087.602,E2 -25087.602} C_VEL
LIN {X 0,Y 129.157,Z 365.393,A -85,B 0,C 180,E1 -25090.945,E2 -25090.945} C_VEL
LIN {X 0,Y 129.416,Z 365.364,A -85,B 0,C 180,E1 -25097.815,E2 -25097.815} C_VEL
LIN {X 0,Y 129.528,Z 365.344,A -85,B 0,C 180,E1 -25100.632,E2 -25100.632} C_VEL
LIN {X 0,Y 130.088,Z 365.274,A -85,B 0,C 180,E1 -25110.001,E2 -25110.001} C_VEL
LIN {X 0,Y 129.529,Z 365.345,A -85,B 0,C 180,E1 -25119.369,E2 -25119.369} C_VEL
LIN {X 0,Y 129.392,Z 365.368,A -85,B 0,C 180,E1 -25122.549,E2 -25122.549} C_VEL
LIN {X 0,Y 129.158,Z 365.394,A -85,B 0,C 180,E1 -25129.056,E2 -25129.056} C_VEL
LIN {X 0,Y 129.106,Z 365.402,A -85,B 0,C 180,E1 -25132.399,E2 -25132.399} C_VEL
LIN {X 0,Y 129.034,Z 365.411,A -85,B 0,C 180,E1 -25139.375,E2 -25139.375} C_VEL
LIN {X 0,Y 128.991,Z 365.412,A -85,B 0,C 180,E1 -25145.19,E2 -25145.19} C_VEL
LIN {X 0,Y 128.95,Z 365.419,A -85,B 0,C 180,E1 -25150.847,E2 -25150.847} C_VEL
LIN {X 0,Y 128.921,Z 365.424,A -85,B 0,C 180,E1 -25155.129,E2 -25155.129} C_VEL
LIN {X 0,Y 129.16,Z 365.5,A -85,B 0,C 180,E1 -25160.842,E2 -25160.842} C_VEL
LIN {X 0,Y 136.827,Z 393.792,A -85,B 0,C 180,E1 -25163.885,E2 -25163.885} C_VEL
LIN {X 0,Y 134.16,Z 450.39,A -85,B 0,C 180,E1 -25169.178,E2 -25169.178} C_VEL
LIN {X 0,Y 133.232,Z 464.524,A -85,B 0,C 180,E1 -25171.013,E2 -25171.013} C_VEL
LIN {X 0,Y 132.025,Z 478.569,A -85,B 0,C 180,E1 -25173.526,E2 -25173.526} C_VEL
LIN {X 0,Y 130.856,Z 490.928,A -85,B 0,C 180,E1 -25176.38,E2 -25176.38} C_VEL
LIN {X 0,Y 129.797,Z 502.771,A -85,B 0,C 180,E1 -25179.809,E2 -25179.809} C_VEL
LIN {X 0,Y 129.056,Z 512.811,A -85,B 0,C 180,E1 -25183.389,E2 -25183.389} C_VEL
LIN {X 0,Y 128.501,Z 523.745,A -85,B 0,C 180,E1 -25188.167,E2 -25188.167} C_VEL
LIN {X 0,Y 128.651,Z 532.807,A -85,B 0,C 180,E1 -25192.962,E2 -25192.962} C_VEL
LIN {X 0,Y 129.566,Z 541.161,A -85,B 0,C 180,E1 -25198.447,E2 -25198.447} C_VEL
LIN {X 0,Y 131.277,Z 547.12,A -85,B 0,C 180,E1 -25203.07,E2 -25203.07} C_VEL
LIN {X 0,Y 133.909,Z 552.013,A -85,B 0,C 180,E1 -25207.541,E2 -25207.541} C_VEL
LIN {X 0,Y 138.62,Z 557.1,A -85,B 0,C 180,E1 -25213.189,E2 -25213.189} C_VEL
LIN {X 0,Y 143.114,Z 559.877,A -85,B 0,C 180,E1 -25217.138,E2 -25217.138} C_VEL
LIN {X 0,Y 150.335,Z 562.282,A -85,B 0,C 180,E1 -25221.963,E2 -25221.963} C_VEL
LIN {X 0,Y 158.564,Z 563.253,A -85,B 0,C 180,E1 -25226.311,E2 -25226.311} C_VEL
LIN {X 0,Y 167.88,Z 562.773,A -85,B 0,C 180,E1 -25230.157,E2 -25230.157} C_VEL
LIN {X 0,Y 177.974,Z 560.798,A -85,B 0,C 180,E1 -25233.564,E2 -25233.564} C_VEL
LIN {X 0,Y 188.784,Z 557.323,A -85,B 0,C 180,E1 -25236.56,E2 -25236.56} C_VEL
LIN {X 0,Y 192.172,Z 555.915,A -85,B 0,C 180,E1 -25237.378,E2 -25237.378} C_VEL
LIN {X 0,Y 192.599,Z 555.924,A -85,B 0,C 180,E1 -25237.924,E2 -25237.924} C_VEL
LIN {X 0,Y 180.166,Z 562.827,A -85,B 0,C 180,E1 -25240.476,E2 -25240.476} C_VEL
LIN {X 0,Y 169.236,Z 567.863,A -85,B 0,C 180,E1 -25243.386,E2 -25243.386} C_VEL
LIN {X 0,Y 161.695,Z 570.757,A -85,B 0,C 180,E1 -25245.937,E2 -25245.937} C_VEL
LIN {X 0,Y 152.587,Z 573.595,A -85,B 0,C 180,E1 -25249.846,E2 -25249.846} C_VEL
LIN {X 0,Y 144.674,Z 575.284,A -85,B 0,C 180,E1 -25254.342,E2 -25254.342} C_VEL
LIN {X 0,Y 138.238,Z 575.859,A -85,B 0,C 180,E1 -25259.442,E2 -25259.442} C_VEL
LIN {X 0,Y 133.557,Z 575.34,A -85,B 0,C 180,E1 -25265.103,E2 -25265.103} C_VEL
LIN {X 0,Y 130.793,Z 573.723,A -85,B 0,C 180,E1 -25271.191,E2 -25271.191} C_VEL
LIN {X 0,Y 130.018,Z 570.934,A -85,B 0,C 180,E1 -25277.512,E2 -25277.512} C_VEL
LIN {X 0,Y 131.306,Z 566.781,A -85,B 0,C 180,E1 -25283.854,E2 -25283.854} C_VEL
LIN {X 0,Y 133.247,Z 562.593,A -85,B 0,C 180,E1 -25288.49,E2 -25288.49} C_VEL
LIN {X 0,Y 134.823,Z 558.354,A -85,B 0,C 180,E1 -25292.032,E2 -25292.032} C_VEL
LIN {X 0,Y 132.428,Z 563.73,A -85,B 0,C 180,E1 -25297.624,E2 -25297.624} C_VEL
LIN {X 0,Y 131.412,Z 567.162,A -85,B 0,C 180,E1 -25302.435,E2 -25302.435} C_VEL
LIN {X 0,Y 130.726,Z 568.365,A -85,B 0,C 180,E1 -25304.951,E2 -25304.951} C_VEL
LIN {X 0,Y 127.505,Z 569.77,A -85,B 0,C 180,E1 -25312.723,E2 -25312.723} C_VEL
LIN {X 0,Y 127.818,Z 570.27,A -85,B 0,C 180,E1 -25315.359,E2 -25315.359} C_VEL
LIN {X 0,Y 128.246,Z 570.502,A -85,B 0,C 180,E1 -25316.212,E2 -25316.212} C_VEL
LIN {X 0,Y 133.643,Z 572.233,A -85,B 0,C 180,E1 -25322.709,E2 -25322.709} C_VEL
LIN {X 0,Y 139.356,Z 572.76,A -85,B 0,C 180,E1 -25327.242,E2 -25327.242} C_VEL
LIN {X 0,Y 147.429,Z 572.509,A -85,B 0,C 180,E1 -25331.865,E2 -25331.865} C_VEL
LIN {X 0,Y 156.82,Z 571.314,A -85,B 0,C 180,E1 -25335.811,E2 -25335.811} C_VEL
LIN {X 0,Y 167.282,Z 569.12,A -85,B 0,C 180,E1 -25339.133,E2 -25339.133} C_VEL
LIN {X 0,Y 169.777,Z 568.459,A -85,B 0,C 180,E1 -25339.806,E2 -25339.806} C_VEL
LIN {X 0,Y 169.329,Z 568.148,A -85,B 0,C 180,E1 -25340.601,E2 -25340.601} C_VEL
LIN {X 0,Y 162.647,Z 567.858,A -85,B 0,C 180,E1 -25342.774,E2 -25342.774} C_VEL
LIN {X 0,Y 152.921,Z 566.287,A -85,B 0,C 180,E1 -25346.529,E2 -25346.529} C_VEL
LIN {X 0,Y 144.264,Z 563.389,A -85,B 0,C 180,E1 -25350.844,E2 -25350.844} C_VEL
LIN {X 0,Y 136.836,Z 559.157,A -85,B 0,C 180,E1 -25355.738,E2 -25355.738} C_VEL
LIN {X 0,Y 130.829,Z 553.469,A -85,B 0,C 180,E1 -25361.196,E2 -25361.196} C_VEL
LIN {X 0,Y 126.35,Z 546.226,A -85,B 0,C 180,E1 -25367.143,E2 -25367.143} C_VEL
LIN {X 0,Y 123.78,Z 538.457,A -85,B 0,C 180,E1 -25372.659,E2 -25372.659} C_VEL
LIN {X 0,Y 122.303,Z 528.944,A -85,B 0,C 180,E1 -25378.352,E2 -25378.352} C_VEL
LIN {X 0,Y 122.17,Z 519.259,A -85,B 0,C 180,E1 -25383.296,E2 -25383.296} C_VEL
LIN {X 0,Y 122.512,Z 507.498,A -85,B 0,C 180,E1 -25388.177,E2 -25388.177} C_VEL
LIN {X 0,Y 123.089,Z 496.646,A -85,B 0,C 180,E1 -25391.866,E2 -25391.866} C_VEL
LIN {X 0,Y 123.951,Z 483.609,A -85,B 0,C 180,E1 -25395.444,E2 -25395.444} C_VEL
LIN {X 0,Y 124.927,Z 469.705,A -85,B 0,C 180,E1 -25398.446,E2 -25398.446} C_VEL
LIN {X 0,Y 125.796,Z 456.043,A -85,B 0,C 180,E1 -25400.649,E2 -25400.649} C_VEL
LIN {X 0,Y 126.82,Z 432.766,A -85,B 0,C 180,E1 -25403.363,E2 -25403.363} C_VEL
LIN {X 0,Y 128.213,Z 390.9,A -85,B 0,C 180,E1 -25407.886,E2 -25407.886} C_VEL
LIN {X 0,Y 122.789,Z 369.346,A -85,B 0,C 180,E1 -25410.242,E2 -25410.242} C_VEL
LIN {X 0,Y 122.216,Z 366.255,A -85,B 0,C 180,E1 -25410.652,E2 -25410.652} C_VEL
LIN {X 0,Y 121.894,Z 366.3,A -85,B 0,C 180,E1 -25416.178,E2 -25416.178} C_VEL
LIN {X 0,Y 121.87,Z 366.304,A -85,B 0,C 180,E1 -25421.437,E2 -25421.437} C_VEL
LIN {X 0,Y 121.882,Z 366.298,A -85,B 0,C 180,E1 -25428.554,E2 -25428.554} C_VEL
LIN {X 0,Y 121.942,Z 366.289,A -85,B 0,C 180,E1 -25434.807,E2 -25434.807} C_VEL
LIN {X 0,Y 121.939,Z 366.295,A -85,B 0,C 180,E1 -25439.826,E2 -25439.826} C_VEL
LIN {X 0,Y 121.981,Z 366.287,A -85,B 0,C 180,E1 -25446.215,E2 -25446.215} C_VEL
LIN {X 0,Y 122.047,Z 366.281,A -85,B 0,C 180,E1 -25449.788,E2 -25449.788} C_VEL
LIN {X 0,Y 122.262,Z 366.256,A -85,B 0,C 180,E1 -25456.707,E2 -25456.707} C_VEL
LIN {X 0,Y 122.454,Z 366.227,A -85,B 0,C 180,E1 -25460.086,E2 -25460.086} C_VEL
LIN {X 0,Y 122.609,Z 366.211,A -85,B 0,C 180,E1 -25466.715,E2 -25466.715} C_VEL
LIN {X 0,Y 123.042,Z 366.151,A -85,B 0,C 180,E1 -25470.001,E2 -25470.001} C_VEL
LIN {X 0,Y 122.454,Z 366.228,A -85,B 0,C 180,E1 -25476.592,E2 -25476.592} C_VEL
LIN {X 0,Y 122.455,Z 366.227,A -85,B 0,C 180,E1 -25479.915,E2 -25479.915} C_VEL
LIN {X 0,Y 122.262,Z 366.255,A -85,B 0,C 180,E1 -25483.294,E2 -25483.294} C_VEL
LIN {X 0,Y 122.048,Z 366.282,A -85,B 0,C 180,E1 -25490.213,E2 -25490.213} C_VEL
LIN {X 0,Y 121.981,Z 366.288,A -85,B 0,C 180,E1 -25493.786,E2 -25493.786} C_VEL
LIN {X 0,Y 121.94,Z 366.296,A -85,B 0,C 180,E1 -25500.175,E2 -25500.175} C_VEL
LIN {X 0,Y 121.911,Z 366.297,A -85,B 0,C 180,E1 -25506.191,E2 -25506.191} C_VEL
LIN {X 0,Y 121.883,Z 366.299,A -85,B 0,C 180,E1 -25511.447,E2 -25511.447} C_VEL
LIN {X 0,Y 121.929,Z 366.295,A -85,B 0,C 180,E1 -25518.533,E2 -25518.533} C_VEL
LIN {X 0,Y 122.075,Z 366.272,A -85,B 0,C 180,E1 -25520.443,E2 -25520.443} C_VEL
LIN {X 0,Y 129.697,Z 395.244,A -85,B 0,C 180,E1 -25523.773,E2 -25523.773} C_VEL
LIN {X 0,Y 127.019,Z 451.212,A -85,B 0,C 180,E1 -25529.333,E2 -25529.333} C_VEL
LIN {X 0,Y 126.056,Z 465.269,A -85,B 0,C 180,E1 -25531.26,E2 -25531.26} C_VEL
LIN {X 0,Y 124.876,Z 478.974,A -85,B 0,C 180,E1 -25533.855,E2 -25533.855} C_VEL
LIN {X 0,Y 123.669,Z 491.744,A -85,B 0,C 180,E1 -25537.004,E2 -25537.004} C_VEL
LIN {X 0,Y 122.649,Z 503.86,A -85,B 0,C 180,E1 -25540.764,E2 -25540.764} C_VEL
LIN {X 0,Y 121.923,Z 514.833,A -85,B 0,C 180,E1 -25544.968,E2 -25544.968} C_VEL
LIN {X 0,Y 121.528,Z 524.44,A -85,B 0,C 180,E1 -25549.462,E2 -25549.462} C_VEL
LIN {X 0,Y 121.947,Z 534.252,A -85,B 0,C 180,E1 -25555.042,E2 -25555.042} C_VEL
LIN {X 0,Y 123.242,Z 542.584,A -85,B 0,C 180,E1 -25560.818,E2 -25560.818} C_VEL
LIN {X 0,Y 125.82,Z 549.315,A -85,B 0,C 180,E1 -25566.416,E2 -25566.416} C_VEL
LIN {X 0,Y 130.28,Z 555.353,A -85,B 0,C 180,E1 -25572.463,E2 -25572.463} C_VEL
LIN {X 0,Y 136.253,Z 559.828,A -85,B 0,C 180,E1 -25578.029,E2 -25578.029} C_VEL
LIN {X 0,Y 143.705,Z 562.792,A -85,B 0,C 180,E1 -25583.034,E2 -25583.034} C_VEL
LIN {X 0,Y 152.198,Z 564.348,A -85,B 0,C 180,E1 -25587.502,E2 -25587.502} C_VEL
LIN {X 0,Y 161.822,Z 564.464,A -85,B 0,C 180,E1 -25591.412,E2 -25591.412} C_VEL
LIN {X 0,Y 172.222,Z 563.103,A -85,B 0,C 180,E1 -25594.843,E2 -25594.843} C_VEL
LIN {X 0,Y 180.59,Z 561.106,A -85,B 0,C 180,E1 -25597.145,E2 -25597.145} C_VEL
LIN {X 0,Y 179.881,Z 561.664,A -85,B 0,C 180,E1 -25597.819,E2 -25597.819} C_VEL
LIN {X 0,Y 169.936,Z 565.979,A -85,B 0,C 180,E1 -25600.083,E2 -25600.083} C_VEL
LIN {X 0,Y 161.769,Z 568.95,A -85,B 0,C 180,E1 -25602.39,E2 -25602.39} C_VEL
LIN {X 0,Y 151.896,Z 571.895,A -85,B 0,C 180,E1 -25606.049,E2 -25606.049} C_VEL
LIN {X 0,Y 142.958,Z 573.692,A -85,B 0,C 180,E1 -25610.275,E2 -25610.275} C_VEL
LIN {X 0,Y 135.415,Z 574.407,A -85,B 0,C 180,E1 -25615.186,E2 -25615.186} C_VEL
LIN {X 0,Y 129.526,Z 574.064,A -85,B 0,C 180,E1 -25620.768,E2 -25620.768} C_VEL
LIN {X 0,Y 125.565,Z 572.657,A -85,B 0,C 180,E1 -25626.933,E2 -25626.933} C_VEL
LIN {X 0,Y 123.651,Z 570.148,A -85,B 0,C 180,E1 -25633.489,E2 -25633.489} C_VEL
LIN {X 0,Y 123.872,Z 566.437,A -85,B 0,C 180,E1 -25640.199,E2 -25640.199} C_VEL
LIN {X 0,Y 125.389,Z 562.657,A -85,B 0,C 180,E1 -25645.177,E2 -25645.177} C_VEL
LIN {X 0,Y 127.105,Z 558.821,A -85,B 0,C 180,E1 -25649.137,E2 -25649.137} C_VEL
LIN {X 0,Y 128.585,Z 554.999,A -85,B 0,C 180,E1 -25652.197,E2 -25652.197} C_VEL
LIN {X 0,Y 126.702,Z 559.179,A -85,B 0,C 180,E1 -25656.369,E2 -25656.369} C_VEL
LIN {X 0,Y 125.068,Z 564.152,A -85,B 0,C 180,E1 -25662.989,E2 -25662.989} C_VEL
LIN {X 0,Y 125.503,Z 567.843,A -85,B 0,C 180,E1 -25669.632,E2 -25669.632} C_VEL
LIN {X 0,Y 128.246,Z 570.502,A -85,B 0,C 180,E1 -25676.212,E2 -25676.212} C_VEL
LIN {X 0,Y 129.368,Z 571.065,A -85,B 0,C 180,E1 -25678.785,E2 -25678.785} C_VEL
